LIN {X 0,Y 466.182,Z 601.705,A -85,B 0,C 180,E1 19756.767,E2 19756.767} C_VEL
LIN {X 0,Y 461.361,Z 693.458,A -85,B 0,C 180,E1 19755.037,E2 19755.037} C_VEL
LIN {X 0,Y 459.117,Z 717.943,A -85,B 0,C 180,E1 19754.37,E2 19754.37} C_VEL
LIN {X 0,Y 456.209,Z 743.457,A -85,B 0,C 180,E1 19753.448,E2 19753.448} C_VEL
LIN {X 0,Y 453.173,Z 765.825,A -85,B 0,C 180,E1 19752.424,E2 19752.424} C_VEL
LIN {X 0,Y 449.498,Z 789.387,A -85,B 0,C 180,E1 19751.096,E2 19751.096} C_VEL
LIN {X 0,Y 445.801,Z 811.052,A -85,B 0,C 180,E1 19749.642,E2 19749.642} C_VEL
LIN {X 0,Y 441.915,Z 831.707,A -85,B 0,C 180,E1 19747.983,E2 19747.983} C_VEL
LIN {X 0,Y 437.866,Z 852.231,A -85,B 0,C 180,E1 19746.062,E2 19746.062} C_VEL
LIN {X 0,Y 434.211,Z 870.106,A -85,B 0,C 180,E1 19744.106,E2 19744.106} C_VEL
LIN {X 0,Y 430.262,Z 889.208,A -85,B 0,C 180,E1 19741.682,E2 19741.682} C_VEL
LIN {X 0,Y 426.966,Z 905.358,A -85,B 0,C 180,E1 19739.304,E2 19739.304} C_VEL
LIN {X 0,Y 423.914,Z 920.881,A -85,B 0,C 180,E1 19736.625,E2 19736.625} C_VEL
LIN {X 0,Y 421.465,Z 934.402,A -85,B 0,C 180,E1 19733.934,E2 19733.934} C_VEL
LIN {X 0,Y 419.512,Z 946.432,A -85,B 0,C 180,E1 19731.094,E2 19731.094} C_VEL
LIN {X 0,Y 418.139,Z 956.77,A -85,B 0,C 180,E1 19728.256,E2 19728.256} C_VEL
LIN {X 0,Y 417.219,Z 965.635,A -85,B 0,C 180,E1 19725.285,E2 19725.285} C_VEL
LIN {X 0,Y 416.734,Z 972.905,A -85,B 0,C 180,E1 19722.33,E2 19722.33} C_VEL
LIN {X 0,Y 416.585,Z 978.694,A -85,B 0,C 180,E1 19719.254,E2 19719.254} C_VEL
LIN {X 0,Y 416.629,Z 982.359,A -85,B 0,C 180,E1 19716.615,E2 19716.615} C_VEL
LIN {X 0,Y 416.736,Z 985.143,A -85,B 0,C 180,E1 19713.577,E2 19713.577} C_VEL
LIN {X 0,Y 416.795,Z 986.147,A -85,B 0,C 180,E1 19710.687,E2 19710.687} C_VEL
LIN {X 0,Y 416.792,Z 985.858,A -85,B 0,C 180,E1 19708.075,E2 19708.075} C_VEL
LIN {X 0,Y 416.657,Z 984.108,A -85,B 0,C 180,E1 19705.044,E2 19705.044} C_VEL
LIN {X 0,Y 416.576,Z 980.619,A -85,B 0,C 180,E1 19701.997,E2 19701.997} C_VEL
LIN {X 0,Y 416.588,Z 976.376,A -85,B 0,C 180,E1 19699.35,E2 19699.35} C_VEL
LIN {X 0,Y 416.89,Z 969.637,A -85,B 0,C 180,E1 19696.122,E2 19696.122} C_VEL
LIN {X 0,Y 417.582,Z 961.789,A -85,B 0,C 180,E1 19693.158,E2 19693.158} C_VEL
LIN {X 0,Y 418.851,Z 951.921,A -85,B 0,C 180,E1 19690.039,E2 19690.039} C_VEL
LIN {X 0,Y 420.695,Z 940.588,A -85,B 0,C 180,E1 19687.059,E2 19687.059} C_VEL
LIN {X 0,Y 423.28,Z 927.489,A -85,B 0,C 180,E1 19684.086,E2 19684.086} C_VEL
LIN {X 0,Y 426.486,Z 912.889,A -85,B 0,C 180,E1 19681.264,E2 19681.264} C_VEL
LIN {X 0,Y 430.666,Z 895.41,A -85,B 0,C 180,E1 19678.351,E2 19678.351} C_VEL
LIN {X 0,Y 435.032,Z 878.269,A -85,B 0,C 180,E1 19675.888,E2 19675.888} C_VEL
LIN {X 0,Y 439.906,Z 859.257,A -85,B 0,C 180,E1 19673.539,E2 19673.539} C_VEL
LIN {X 0,Y 445.064,Z 839.529,A -85,B 0,C 180,E1 19671.428,E2 19671.428} C_VEL
LIN {X 0,Y 450.442,Z 818.443,A -85,B 0,C 180,E1 19669.512,E2 19669.512} C_VEL
LIN {X 0,Y 455.993,Z 795.957,A -85,B 0,C 180,E1 19667.772,E2 19667.772} C_VEL
LIN {X 0,Y 461.455,Z 772.834,A -85,B 0,C 180,E1 19666.273,E2 19666.273} C_VEL
LIN {X 0,Y 466.711,Z 748.74,A -85,B 0,C 180,E1 19664.991,E2 19664.991} C_VEL
LIN {X 0,Y 471.508,Z 724.263,A -85,B 0,C 180,E1 19663.949,E2 19663.949} C_VEL
LIN {X 0,Y 476.08,Z 697.875,A -85,B 0,C 180,E1 19663.088,E2 19663.088} C_VEL
LIN {X 0,Y 481.22,Z 660.217,A -85,B 0,C 180,E1 19662.172,E2 19662.172} C_VEL
LIN {X 0,Y 489.533,Z 604.335,A -85,B 0,C 180,E1 19660.843,E2 19660.843} C_VEL
LIN {X 0,Y 500.202,Z 547.443,A -85,B 0,C 180,E1 19659.451,E2 19659.451} C_VEL
LIN {X 0,Y 508.93,Z 508.11,A -85,B 0,C 180,E1 19658.468,E2 19658.468} C_VEL
LIN {X 0,Y 504.603,Z 526.167,A -85,B 0,C 180,E1 19657.559,E2 19657.559} C_VEL
LIN {X 0,Y 481.706,Z 630.182,A -85,B 0,C 180,E1 19654.492,E2 19654.492} C_VEL
LIN {X 0,Y 469.101,Z 693.847,A -85,B 0,C 180,E1 19652.444,E2 19652.444} C_VEL
LIN {X 0,Y 463.766,Z 717.456,A -85,B 0,C 180,E1 19651.45,E2 19651.45} C_VEL
LIN {X 0,Y 458.09,Z 740.922,A -85,B 0,C 180,E1 19650.185,E2 19650.185} C_VEL
LIN {X 0,Y 452.388,Z 763.754,A -85,B 0,C 180,E1 19648.661,E2 19648.661} C_VEL
LIN {X 0,Y 447.011,Z 785.108,A -85,B 0,C 180,E1 19646.934,E2 19646.934} C_VEL
LIN {X 0,Y 442.238,Z 804.171,A -85,B 0,C 180,E1 19645.083,E2 19645.083} C_VEL
LIN {X 0,Y 437.83,Z 821.686,A -85,B 0,C 180,E1 19643.058,E2 19643.058} C_VEL
LIN {X 0,Y 433.913,Z 837.047,A -85,B 0,C 180,E1 19640.927,E2 19640.927} C_VEL
LIN {X 0,Y 430.445,Z 850.31,A -85,B 0,C 180,E1 19638.697,E2 19638.697} C_VEL
LIN {X 0,Y 427.606,Z 860.933,A -85,B 0,C 180,E1 19636.519,E2 19636.519} C_VEL
LIN {X 0,Y 425.193,Z 869.743,A -85,B 0,C 180,E1 19634.295,E2 19634.295} C_VEL
LIN {X 0,Y 423.039,Z 877.204,A -85,B 0,C 180,E1 19631.867,E2 19631.867} C_VEL
LIN {X 0,Y 421.42,Z 882.367,A -85,B 0,C 180,E1 19629.56,E2 19629.56} C_VEL
LIN {X 0,Y 420.191,Z 885.911,A -85,B 0,C 180,E1 19627.245,E2 19627.245} C_VEL
LIN {X 0,Y 419.213,Z 887.887,A -85,B 0,C 180,E1 19624.789,E2 19624.789} C_VEL
LIN {X 0,Y 418.581,Z 888.17,A -85,B 0,C 180,E1 19622.464,E2 19622.464} C_VEL
LIN {X 0,Y 418.161,Z 886.727,A -85,B 0,C 180,E1 19620,E2 19620} C_VEL
LIN {X 0,Y 417.948,Z 883.54,A -85,B 0,C 180,E1 19617.532,E2 19617.532} C_VEL
LIN {X 0,Y 417.955,Z 878.555,A -85,B 0,C 180,E1 19615.059,E2 19615.059} C_VEL
LIN {X 0,Y 418.197,Z 871.701,A -85,B 0,C 180,E1 19612.582,E2 19612.582} C_VEL
LIN {X 0,Y 418.711,Z 862.825,A -85,B 0,C 180,E1 19610.099,E2 19610.099} C_VEL
LIN {X 0,Y 419.516,Z 852.331,A -85,B 0,C 180,E1 19607.745,E2 19607.745} C_VEL
LIN {X 0,Y 420.579,Z 840.438,A -85,B 0,C 180,E1 19605.544,E2 19605.544} C_VEL
LIN {X 0,Y 421.988,Z 826.127,A -85,B 0,C 180,E1 19603.339,E2 19603.339} C_VEL
LIN {X 0,Y 423.658,Z 810.108,A -85,B 0,C 180,E1 19601.278,E2 19601.278} C_VEL
LIN {X 0,Y 425.556,Z 792.28,A -85,B 0,C 180,E1 19599.363,E2 19599.363} C_VEL
LIN {X 0,Y 427.535,Z 773.248,A -85,B 0,C 180,E1 19597.663,E2 19597.663} C_VEL
LIN {X 0,Y 429.463,Z 754.068,A -85,B 0,C 180,E1 19596.247,E2 19596.247} C_VEL
LIN {X 0,Y 431.425,Z 733.007,A -85,B 0,C 180,E1 19594.986,E2 19594.986} C_VEL
LIN {X 0,Y 433.222,Z 711.178,A -85,B 0,C 180,E1 19593.953,E2 19593.953} C_VEL
LIN {X 0,Y 434.895,Z 687.679,A -85,B 0,C 180,E1 19593.121,E2 19593.121} C_VEL
LIN {X 0,Y 437.042,Z 646.566,A -85,B 0,C 180,E1 19592.122,E2 19592.122} C_VEL
LIN {X 0,Y 444.712,Z 506.021,A -85,B 0,C 180,E1 19588.907,E2 19588.907} C_VEL
LIN {X 0,Y 439.779,Z 438.733,A -85,B 0,C 180,E1 19586.694,E2 19586.694} C_VEL
LIN {X 0,Y 445.969,Z 387.644,A -85,B 0,C 180,E1 19582.511,E2 19582.511} C_VEL
LIN {X 0,Y 451.691,Z 344.172,A -85,B 0,C 180,E1 19578.936,E2 19578.936} C_VEL
LIN {X 0,Y 453.675,Z 344.144,A -85,B 0,C 180,E1 19578.609,E2 19578.609} C_VEL
LIN {X 0,Y 456.593,Z 342.501,A -85,B 0,C 180,E1 19578.262,E2 19578.262} C_VEL
LIN {X 0,Y 459.898,Z 339.563,A -85,B 0,C 180,E1 19577.96,E2 19577.96} C_VEL
LIN {X 0,Y 463.43,Z 338.215,A -85,B 0,C 180,E1 19577.52,E2 19577.52} C_VEL
LIN {X 0,Y 468.257,Z 334.771,A -85,B 0,C 180,E1 19577.064,E2 19577.064} C_VEL
LIN {X 0,Y 472.208,Z 333.263,A -85,B 0,C 180,E1 19576.6,E2 19576.6} C_VEL
LIN {X 0,Y 476.586,Z 346.018,A -85,B 0,C 180,E1 19574.994,E2 19574.994} C_VEL
LIN {X 0,Y 476.081,Z 370.363,A -85,B 0,C 180,E1 19573.293,E2 19573.293} C_VEL
LIN {X 0,Y 470.702,Z 395.368,A -85,B 0,C 180,E1 19572.381,E2 19572.381} C_VEL
LIN {X 0,Y 466.885,Z 477.849,A -85,B 0,C 180,E1 19571.021,E2 19571.021} C_VEL
LIN {X 0,Y 462.789,Z 540.682,A -85,B 0,C 180,E1 19569.779,E2 19569.779} C_VEL
LIN {X 0,Y 457.359,Z 607.896,A -85,B 0,C 180,E1 19568.227,E2 19568.227} C_VEL
LIN {X 0,Y 453.808,Z 652.838,A -85,B 0,C 180,E1 19567.008,E2 19567.008} C_VEL
LIN {X 0,Y 452.145,Z 676.013,A -85,B 0,C 180,E1 19566.219,E2 19566.219} C_VEL
LIN {X 0,Y 450.073,Z 696.948,A -85,B 0,C 180,E1 19565.284,E2 19565.284} C_VEL
LIN {X 0,Y 447.372,Z 718.396,A -85,B 0,C 180,E1 19564.073,E2 19564.073} C_VEL
LIN {X 0,Y 444.251,Z 739.171,A -85,B 0,C 180,E1 19562.619,E2 19562.619} C_VEL
LIN {X 0,Y 440.936,Z 758.361,A -85,B 0,C 180,E1 19560.992,E2 19560.992} C_VEL
LIN {X 0,Y 438.931,Z 764.725,A -85,B 0,C 180,E1 19560.467,E2 19560.467} C_VEL
LIN {X 0,Y 430.735,Z 780.584,A -85,B 0,C 180,E1 19559.246,E2 19559.246} C_VEL
LIN {X 0,Y 428.649,Z 786.403,A -85,B 0,C 180,E1 19558.626,E2 19558.626} C_VEL
LIN {X 0,Y 425.203,Z 802.108,A -85,B 0,C 180,E1 19556.538,E2 19556.538} C_VEL
LIN {X 0,Y 421.843,Z 816.908,A -85,B 0,C 180,E1 19554.209,E2 19554.209} C_VEL
LIN {X 0,Y 418.786,Z 830.224,A -85,B 0,C 180,E1 19551.72,E2 19551.72} C_VEL
LIN {X 0,Y 415.99,Z 842.599,A -85,B 0,C 180,E1 19548.935,E2 19548.935} C_VEL
LIN {X 0,Y 413.787,Z 852.799,A -85,B 0,C 180,E1 19546.134,E2 19546.134} C_VEL
LIN {X 0,Y 412.078,Z 861.435,A -85,B 0,C 180,E1 19543.185,E2 19543.185} C_VEL
LIN {X 0,Y 410.917,Z 867.862,A -85,B 0,C 180,E1 19540.374,E2 19540.374} C_VEL
LIN {X 0,Y 410.156,Z 872.891,A -85,B 0,C 180,E1 19537.424,E2 19537.424} C_VEL
LIN {X 0,Y 409.729,Z 876.243,A -85,B 0,C 180,E1 19534.479,E2 19534.479} C_VEL
LIN {X 0,Y 409.54,Z 877.981,A -85,B 0,C 180,E1 19531.539,E2 19531.539} C_VEL
LIN {X 0,Y 409.523,Z 878.039,A -85,B 0,C 180,E1 19528.741,E2 19528.741} C_VEL
LIN {X 0,Y 409.692,Z 876.537,A -85,B 0,C 180,E1 19525.801,E2 19525.801} C_VEL
LIN {X 0,Y 410.094,Z 873.424,A -85,B 0,C 180,E1 19522.857,E2 19522.857} C_VEL
LIN {X 0,Y 410.768,Z 868.937,A -85,B 0,C 180,E1 19520.048,E2 19520.048} C_VEL
LIN {X 0,Y 411.91,Z 862.424,A -85,B 0,C 180,E1 19517.096,E2 19517.096} C_VEL
LIN {X 0,Y 413.462,Z 854.365,A -85,B 0,C 180,E1 19514.26,E2 19514.26} C_VEL
LIN {X 0,Y 415.547,Z 844.595,A -85,B 0,C 180,E1 19511.481,E2 19511.481} C_VEL
LIN {X 0,Y 418.086,Z 833.296,A -85,B 0,C 180,E1 19508.83,E2 19508.83} C_VEL
LIN {X 0,Y 421.02,Z 820.573,A -85,B 0,C 180,E1 19506.337,E2 19506.337} C_VEL
LIN {X 0,Y 424.266,Z 806.441,A -85,B 0,C 180,E1 19504.001,E2 19504.001} C_VEL
LIN {X 0,Y 427.748,Z 790.854,A -85,B 0,C 180,E1 19501.824,E2 19501.824} C_VEL
LIN {X 0,Y 431.38,Z 773.694,A -85,B 0,C 180,E1 19499.803,E2 19499.803} C_VEL
LIN {X 0,Y 434.929,Z 755.568,A -85,B 0,C 180,E1 19498.008,E2 19498.008} C_VEL
LIN {X 0,Y 438.301,Z 736.243,A -85,B 0,C 180,E1 19496.412,E2 19496.412} C_VEL
LIN {X 0,Y 441.375,Z 715.92,A -85,B 0,C 180,E1 19495.03,E2 19495.03} C_VEL
LIN {X 0,Y 443.968,Z 695.234,A -85,B 0,C 180,E1 19493.891,E2 19493.891} C_VEL
LIN {X 0,Y 446.008,Z 674.403,A -85,B 0,C 180,E1 19492.983,E2 19492.983} C_VEL
LIN {X 0,Y 447.966,Z 647.329,A -85,B 0,C 180,E1 19492.093,E2 19492.093} C_VEL
LIN {X 0,Y 452.25,Z 596.981,A -85,B 0,C 180,E1 19490.753,E2 19490.753} C_VEL
LIN {X 0,Y 457.54,Z 531.945,A -85,B 0,C 180,E1 19489.27,E2 19489.27} C_VEL
LIN {X 0,Y 461.65,Z 467.541,A -85,B 0,C 180,E1 19488.024,E2 19488.024} C_VEL
LIN {X 0,Y 465.122,Z 396.05,A -85,B 0,C 180,E1 19486.831,E2 19486.831} C_VEL
LIN {X 0,Y 470.511,Z 371.711,A -85,B 0,C 180,E1 19485.914,E2 19485.914} C_VEL
LIN {X 0,Y 470.855,Z 349.322,A -85,B 0,C 180,E1 19484.319,E2 19484.319} C_VEL
LIN {X 0,Y 463.855,Z 330.038,A -85,B 0,C 180,E1 19481.766,E2 19481.766} C_VEL
LIN {X 0,Y 456.491,Z 312.145,A -85,B 0,C 180,E1 19479.112,E2 19479.112} C_VEL
LIN {X 0,Y 448.714,Z 295.881,A -85,B 0,C 180,E1 19476.445,E2 19476.445} C_VEL
LIN {X 0,Y 441.192,Z 281.498,A -85,B 0,C 180,E1 19473.806,E2 19473.806} C_VEL
LIN {X 0,Y 434.542,Z 270.327,A -85,B 0,C 180,E1 19471.489,E2 19471.489} C_VEL
LIN {X 0,Y 429.661,Z 262.251,A -85,B 0,C 180,E1 19469.715,E2 19469.715} C_VEL
LIN {X 0,Y 426.904,Z 258.059,A -85,B 0,C 180,E1 19468.695,E2 19468.695} C_VEL
LIN {X 0,Y 423.194,Z 252.399,A -85,B 0,C 180,E1 19467.282,E2 19467.282} C_VEL
LIN {X 0,Y 419.793,Z 247.902,A -85,B 0,C 180,E1 19465.993,E2 19465.993} C_VEL
LIN {X 0,Y 418.942,Z 246.069,A -85,B 0,C 180,E1 19465.594,E2 19465.594} C_VEL
LIN {X 0,Y 416.059,Z 242.908,A -85,B 0,C 180,E1 19464.492,E2 19464.492} C_VEL
LIN {X 0,Y 414.671,Z 240.056,A -85,B 0,C 180,E1 19463.822,E2 19463.822} C_VEL
LIN {X 0,Y 411.827,Z 237.422,A -85,B 0,C 180,E1 19462.709,E2 19462.709} C_VEL
LIN {X 0,Y 410.633,Z 234.295,A -85,B 0,C 180,E1 19462.024,E2 19462.024} C_VEL
LIN {X 0,Y 410.594,Z 234.03,A -85,B 0,C 180,E1 19458.162,E2 19458.162} C_VEL
LIN {X 0,Y 410.604,Z 234.058,A -85,B 0,C 180,E1 19454.238,E2 19454.238} C_VEL
LIN {X 0,Y 410.596,Z 234.057,A -85,B 0,C 180,E1 19450.24,E2 19450.24} C_VEL
LIN {X 0,Y 410.596,Z 234.027,A -85,B 0,C 180,E1 19446.291,E2 19446.291} C_VEL
LIN {X 0,Y 410.601,Z 234.083,A -85,B 0,C 180,E1 19442.373,E2 19442.373} C_VEL
LIN {X 0,Y 410.597,Z 234.031,A -85,B 0,C 180,E1 19438.465,E2 19438.465} C_VEL
LIN {X 0,Y 410.599,Z 234.046,A -85,B 0,C 180,E1 19434.55,E2 19434.55} C_VEL
LIN {X 0,Y 410.602,Z 234.061,A -85,B 0,C 180,E1 19430.61,E2 19430.61} C_VEL
LIN {X 0,Y 410.605,Z 234.083,A -85,B 0,C 180,E1 19426.624,E2 19426.624} C_VEL
LIN {X 0,Y 410.601,Z 234.084,A -85,B 0,C 180,E1 19422.717,E2 19422.717} C_VEL
LIN {X 0,Y 410.633,Z 234.282,A -85,B 0,C 180,E1 19422.462,E2 19422.462} C_VEL
LIN {X 0,Y 411.874,Z 237.541,A -85,B 0,C 180,E1 19421.75,E2 19421.75} C_VEL
LIN {X 0,Y 413.191,Z 239.4,A -85,B 0,C 180,E1 19421.225,E2 19421.225} C_VEL
LIN {X 0,Y 415.204,Z 243.299,A -85,B 0,C 180,E1 19420.297,E2 19420.297} C_VEL
LIN {X 0,Y 420.886,Z 254.249,A -85,B 0,C 180,E1 19417.807,E2 19417.807} C_VEL
LIN {X 0,Y 427.8,Z 267.468,A -85,B 0,C 180,E1 19414.973,E2 19414.973} C_VEL
LIN {X 0,Y 436.306,Z 284.141,A -85,B 0,C 180,E1 19411.68,E2 19411.68} C_VEL
LIN {X 0,Y 446.297,Z 304.362,A -85,B 0,C 180,E1 19408.08,E2 19408.08} C_VEL
LIN {X 0,Y 456.718,Z 326.072,A -85,B 0,C 180,E1 19404.634,E2 19404.634} C_VEL
LIN {X 0,Y 474.355,Z 353.885,A -85,B 0,C 180,E1 19402.032,E2 19402.032} C_VEL
LIN {X 0,Y 474.205,Z 360.312,A -85,B 0,C 180,E1 19401.883,E2 19401.883} C_VEL
LIN {X 0,Y 459.21,Z 606.522,A -85,B 0,C 180,E1 19397.216,E2 19397.216} C_VEL
LIN {X 0,Y 454.457,Z 693.43,A -85,B 0,C 180,E1 19395.543,E2 19395.543} C_VEL
LIN {X 0,Y 452.163,Z 717.773,A -85,B 0,C 180,E1 19394.869,E2 19394.869} C_VEL
LIN {X 0,Y 449.295,Z 742.351,A -85,B 0,C 180,E1 19393.975,E2 19393.975} C_VEL
LIN {X 0,Y 446.278,Z 764.081,A -85,B 0,C 180,E1 19392.975,E2 19392.975} C_VEL
LIN {X 0,Y 442.507,Z 787.894,A -85,B 0,C 180,E1 19391.63,E2 19391.63} C_VEL
LIN {X 0,Y 438.714,Z 809.559,A -85,B 0,C 180,E1 19390.165,E2 19390.165} C_VEL
LIN {X 0,Y 434.774,Z 830.163,A -85,B 0,C 180,E1 19388.501,E2 19388.501} C_VEL
LIN {X 0,Y 430.744,Z 850.203,A -85,B 0,C 180,E1 19386.625,E2 19386.625} C_VEL
LIN {X 0,Y 426.766,Z 869.103,A -85,B 0,C 180,E1 19384.541,E2 19384.541} C_VEL
LIN {X 0,Y 422.811,Z 887.794,A -85,B 0,C 180,E1 19382.147,E2 19382.147} C_VEL
LIN {X 0,Y 419.509,Z 903.423,A -85,B 0,C 180,E1 19379.82,E2 19379.82} C_VEL
LIN {X 0,Y 416.377,Z 918.925,A -85,B 0,C 180,E1 19377.146,E2 19377.146} C_VEL
LIN {X 0,Y 413.922,Z 931.913,A -85,B 0,C 180,E1 19374.55,E2 19374.55} C_VEL
LIN {X 0,Y 411.744,Z 944.833,A -85,B 0,C 180,E1 19371.512,E2 19371.512} C_VEL
LIN {X 0,Y 410.284,Z 955.269,A -85,B 0,C 180,E1 19368.618,E2 19368.618} C_VEL
LIN {X 0,Y 409.272,Z 964.688,A -85,B 0,C 180,E1 19365.444,E2 19365.444} C_VEL
LIN {X 0,Y 408.776,Z 971.983,A -85,B 0,C 180,E1 19362.43,E2 19362.43} C_VEL
LIN {X 0,Y 408.629,Z 977.786,A -85,B 0,C 180,E1 19359.294,E2 19359.294} C_VEL
LIN {X 0,Y 408.681,Z 981.444,A -85,B 0,C 180,E1 19356.603,E2 19356.603} C_VEL
LIN {X 0,Y 408.797,Z 984.212,A -85,B 0,C 180,E1 19353.506,E2 19353.506} C_VEL
LIN {X 0,Y 408.855,Z 985.183,A -85,B 0,C 180,E1 19350.56,E2 19350.56} C_VEL
LIN {X 0,Y 408.837,Z 984.862,A -85,B 0,C 180,E1 19347.898,E2 19347.898} C_VEL
LIN {X 0,Y 408.69,Z 983.057,A -85,B 0,C 180,E1 19344.806,E2 19344.806} C_VEL
LIN {X 0,Y 408.594,Z 979.51,A -85,B 0,C 180,E1 19341.698,E2 19341.698} C_VEL
LIN {X 0,Y 408.613,Z 975.041,A -85,B 0,C 180,E1 19338.892,E2 19338.892} C_VEL
LIN {X 0,Y 408.992,Z 968.066,A -85,B 0,C 180,E1 19335.56,E2 19335.56} C_VEL
LIN {X 0,Y 409.782,Z 960.115,A -85,B 0,C 180,E1 19332.535,E2 19332.535} C_VEL
LIN {X 0,Y 411.287,Z 949.569,A -85,B 0,C 180,E1 19329.21,E2 19329.21} C_VEL
LIN {X 0,Y 413.253,Z 938.67,A -85,B 0,C 180,E1 19326.319,E2 19326.319} C_VEL
LIN {X 0,Y 416.402,Z 923.909,A -85,B 0,C 180,E1 19322.983,E2 19322.983} C_VEL
LIN {X 0,Y 419.914,Z 909.28,A -85,B 0,C 180,E1 19320.154,E2 19320.154} C_VEL
LIN {X 0,Y 424.304,Z 892.298,A -85,B 0,C 180,E1 19317.34,E2 19317.34} C_VEL
LIN {X 0,Y 429.296,Z 873.956,A -85,B 0,C 180,E1 19314.716,E2 19314.716} C_VEL
LIN {X 0,Y 434.639,Z 854.657,A -85,B 0,C 180,E1 19312.354,E2 19312.354} C_VEL
LIN {X 0,Y 440.371,Z 833.928,A -85,B 0,C 180,E1 19310.186,E2 19310.186} C_VEL
LIN {X 0,Y 445.99,Z 813.441,A -85,B 0,C 180,E1 19308.337,E2 19308.337} C_VEL
LIN {X 0,Y 451.965,Z 790.62,A -85,B 0,C 180,E1 19306.613,E2 19306.613} C_VEL
LIN {X 0,Y 457.815,Z 767.151,A -85,B 0,C 180,E1 19305.134,E2 19305.134} C_VEL
LIN {X 0,Y 463.428,Z 743.115,A -85,B 0,C 180,E1 19303.893,E2 19303.893} C_VEL
LIN {X 0,Y 468.675,Z 718.317,A -85,B 0,C 180,E1 19302.875,E2 19302.875} C_VEL
LIN {X 0,Y 473.177,Z 693.617,A -85,B 0,C 180,E1 19302.1,E2 19302.1} C_VEL
LIN {X 0,Y 485.132,Z 617.626,A -85,B 0,C 180,E1 19300.249,E2 19300.249} C_VEL
LIN {X 0,Y 496.148,Z 562.189,A -85,B 0,C 180,E1 19298.884,E2 19298.884} C_VEL
LIN {X 0,Y 502.171,Z 535.812,A -85,B 0,C 180,E1 19298.223,E2 19298.223} C_VEL
LIN {X 0,Y 478.06,Z 639.781,A -85,B 0,C 180,E1 19295.149,E2 19295.149} C_VEL
LIN {X 0,Y 466.558,Z 693.913,A -85,B 0,C 180,E1 19293.393,E2 19293.393} C_VEL
LIN {X 0,Y 460.795,Z 717.287,A -85,B 0,C 180,E1 19292.41,E2 19292.41} C_VEL
LIN {X 0,Y 454.74,Z 739.998,A -85,B 0,C 180,E1 19291.186,E2 19291.186} C_VEL
LIN {X 0,Y 448.459,Z 762.678,A -85,B 0,C 180,E1 19289.668,E2 19289.668} C_VEL
LIN {X 0,Y 442.189,Z 785.109,A -85,B 0,C 180,E1 19287.836,E2 19287.836} C_VEL
LIN {X 0,Y 436.82,Z 804.476,A -85,B 0,C 180,E1 19285.926,E2 19285.926} C_VEL
LIN {X 0,Y 432.024,Z 821.806,A -85,B 0,C 180,E1 19283.893,E2 19283.893} C_VEL
LIN {X 0,Y 427.866,Z 836.688,A -85,B 0,C 180,E1 19281.813,E2 19281.813} C_VEL
LIN {X 0,Y 424.085,Z 850.143,A -85,B 0,C 180,E1 19279.561,E2 19279.561} C_VEL
LIN {X 0,Y 420.685,Z 861.897,A -85,B 0,C 180,E1 19277.141,E2 19277.141} C_VEL
LIN {X 0,Y 417.846,Z 871.334,A -85,B 0,C 180,E1 19274.694,E2 19274.694} C_VEL
LIN {X 0,Y 415.638,Z 878.281,A -85,B 0,C 180,E1 19272.363,E2 19272.363} C_VEL
LIN {X 0,Y 413.877,Z 883.502,A -85,B 0,C 180,E1 19270.017,E2 19270.017} C_VEL
LIN {X 0,Y 412.447,Z 887.202,A -85,B 0,C 180,E1 19267.522,E2 19267.522} C_VEL
LIN {X 0,Y 411.394,Z 889.136,A -85,B 0,C 180,E1 19265.02,E2 19265.02} C_VEL
LIN {X 0,Y 410.666,Z 889.291,A -85,B 0,C 180,E1 19262.512,E2 19262.512} C_VEL
LIN {X 0,Y 410.24,Z 887.847,A -85,B 0,C 180,E1 19260.14,E2 19260.14} C_VEL
LIN {X 0,Y 410.002,Z 884.604,A -85,B 0,C 180,E1 19257.624,E2 19257.624} C_VEL
LIN {X 0,Y 409.997,Z 879.569,A -85,B 0,C 180,E1 19255.103,E2 19255.103} C_VEL
LIN {X 0,Y 410.237,Z 872.646,A -85,B 0,C 180,E1 19252.578,E2 19252.578} C_VEL
LIN {X 0,Y 410.759,Z 863.693,A -85,B 0,C 180,E1 19250.047,E2 19250.047} C_VEL
LIN {X 0,Y 411.582,Z 853.184,A -85,B 0,C 180,E1 19247.656,E2 19247.656} C_VEL
LIN {X 0,Y 412.682,Z 841.23,A -85,B 0,C 180,E1 19245.405,E2 19245.405} C_VEL
LIN {X 0,Y 414.082,Z 827.361,A -85,B 0,C 180,E1 19243.228,E2 19243.228} C_VEL
LIN {X 0,Y 415.785,Z 811.363,A -85,B 0,C 180,E1 19241.128,E2 19241.128} C_VEL
LIN {X 0,Y 417.725,Z 793.581,A -85,B 0,C 180,E1 19239.178,E2 19239.178} C_VEL
LIN {X 0,Y 419.747,Z 774.635,A -85,B 0,C 180,E1 19237.448,E2 19237.448} C_VEL
LIN {X 0,Y 421.818,Z 754.622,A -85,B 0,C 180,E1 19235.939,E2 19235.939} C_VEL
LIN {X 0,Y 423.846,Z 733.462,A -85,B 0,C 180,E1 19234.648,E2 19234.648} C_VEL
LIN {X 0,Y 425.613,Z 712.677,A -85,B 0,C 180,E1 19233.639,E2 19233.639} C_VEL
LIN {X 0,Y 427.276,Z 690.14,A -85,B 0,C 180,E1 19232.808,E2 19232.808} C_VEL
LIN {X 0,Y 429.095,Z 657.974,A -85,B 0,C 180,E1 19231.976,E2 19231.976} C_VEL
LIN {X 0,Y 437.616,Z 506.725,A -85,B 0,C 180,E1 19228.426,E2 19228.426} C_VEL
LIN {X 0,Y 432.779,Z 437.458,A -85,B 0,C 180,E1 19226.085,E2 19226.085} C_VEL
LIN {X 0,Y 439.247,Z 386.125,A -85,B 0,C 180,E1 19221.827,E2 19221.827} C_VEL
LIN {X 0,Y 443.283,Z 356.55,A -85,B 0,C 180,E1 19219.359,E2 19219.359} C_VEL
LIN {X 0,Y 445.261,Z 356.47,A -85,B 0,C 180,E1 19219.025,E2 19219.025} C_VEL
LIN {X 0,Y 448.955,Z 354.156,A -85,B 0,C 180,E1 19218.588,E2 19218.588} C_VEL
LIN {X 0,Y 451.823,Z 351.613,A -85,B 0,C 180,E1 19218.317,E2 19218.317} C_VEL
LIN {X 0,Y 455.703,Z 349.897,A -85,B 0,C 180,E1 19217.823,E2 19217.823} C_VEL
LIN {X 0,Y 460.446,Z 346.36,A -85,B 0,C 180,E1 19217.349,E2 19217.349} C_VEL
LIN {X 0,Y 465.632,Z 343.618,A -85,B 0,C 180,E1 19216.763,E2 19216.763} C_VEL
LIN {X 0,Y 468.15,Z 341.884,A -85,B 0,C 180,E1 19216.527,E2 19216.527} C_VEL
LIN {X 0,Y 470.899,Z 349.839,A -85,B 0,C 180,E1 19215.516,E2 19215.516} C_VEL
LIN {X 0,Y 470.365,Z 372.226,A -85,B 0,C 180,E1 19213.953,E2 19213.953} C_VEL
LIN {X 0,Y 464.775,Z 398.05,A -85,B 0,C 180,E1 19213.014,E2 19213.014} C_VEL
LIN {X 0,Y 460.852,Z 480.196,A -85,B 0,C 180,E1 19211.649,E2 19211.649} C_VEL
LIN {X 0,Y 456.69,Z 542.095,A -85,B 0,C 180,E1 19210.412,E2 19210.412} C_VEL
LIN {X 0,Y 451.226,Z 607.78,A -85,B 0,C 180,E1 19208.878,E2 19208.878} C_VEL
LIN {X 0,Y 447.491,Z 653.023,A -85,B 0,C 180,E1 19207.635,E2 19207.635} C_VEL
LIN {X 0,Y 445.668,Z 677.543,A -85,B 0,C 180,E1 19206.792,E2 19206.792} C_VEL
LIN {X 0,Y 443.448,Z 699.052,A -85,B 0,C 180,E1 19205.812,E2 19205.812} C_VEL
LIN {X 0,Y 440.746,Z 719.67,A -85,B 0,C 180,E1 19204.628,E2 19204.628} C_VEL
LIN {X 0,Y 437.713,Z 739.284,A -85,B 0,C 180,E1 19203.247,E2 19203.247} C_VEL
LIN {X 0,Y 434.389,Z 758.036,A -85,B 0,C 180,E1 19201.656,E2 19201.656} C_VEL
LIN {X 0,Y 430.869,Z 775.879,A -85,B 0,C 180,E1 19199.853,E2 19199.853} C_VEL
LIN {X 0,Y 428.649,Z 786.403,A -85,B 0,C 180,E1 19198.626,E2 19198.626} C_VEL
LIN {X 0,Y 426.569,Z 792.199,A -85,B 0,C 180,E1 19197.982,E2 19197.982} C_VEL
LIN {X 0,Y 418.163,Z 806.503,A -85,B 0,C 180,E1 19196.446,E2 19196.446} C_VEL
LIN {X 0,Y 416.054,Z 811.677,A -85,B 0,C 180,E1 19195.707,E2 19195.707} C_VEL
LIN {X 0,Y 412.727,Z 825.579,A -85,B 0,C 180,E1 19193.259,E2 19193.259} C_VEL
LIN {X 0,Y 409.828,Z 837.724,A -85,B 0,C 180,E1 19190.718,E2 19190.718} C_VEL
LIN {X 0,Y 407.198,Z 848.973,A -85,B 0,C 180,E1 19187.875,E2 19187.875} C_VEL
LIN {X 0,Y 405.09,Z 858.595,A -85,B 0,C 180,E1 19184.875,E2 19184.875} C_VEL
LIN {X 0,Y 403.628,Z 865.866,A -85,B 0,C 180,E1 19182.011,E2 19182.011} C_VEL
LIN {X 0,Y 402.636,Z 871.479,A -85,B 0,C 180,E1 19179.145,E2 19179.145} C_VEL
LIN {X 0,Y 402.009,Z 875.701,A -85,B 0,C 180,E1 19176.14,E2 19176.14} C_VEL
LIN {X 0,Y 401.697,Z 878.215,A -85,B 0,C 180,E1 19173.282,E2 19173.282} C_VEL
LIN {X 0,Y 401.58,Z 879.177,A -85,B 0,C 180,E1 19170.285,E2 19170.285} C_VEL
LIN {X 0,Y 401.639,Z 878.588,A -85,B 0,C 180,E1 19167.432,E2 19167.432} C_VEL
LIN {X 0,Y 401.919,Z 876.416,A -85,B 0,C 180,E1 19164.432,E2 19164.432} C_VEL
LIN {X 0,Y 402.47,Z 872.618,A -85,B 0,C 180,E1 19161.427,E2 19161.427} C_VEL
LIN {X 0,Y 403.427,Z 867.074,A -85,B 0,C 180,E1 19158.419,E2 19158.419} C_VEL
LIN {X 0,Y 404.801,Z 859.988,A -85,B 0,C 180,E1 19155.53,E2 19155.53} C_VEL
LIN {X 0,Y 406.685,Z 851.263,A -85,B 0,C 180,E1 19152.693,E2 19152.693} C_VEL
LIN {X 0,Y 409.166,Z 840.507,A -85,B 0,C 180,E1 19149.845,E2 19149.845} C_VEL
LIN {X 0,Y 412.106,Z 828.21,A -85,B 0,C 180,E1 19147.157,E2 19147.157} C_VEL
LIN {X 0,Y 415.446,Z 814.375,A -85,B 0,C 180,E1 19144.633,E2 19144.633} C_VEL
LIN {X 0,Y 418.979,Z 799.456,A -85,B 0,C 180,E1 19142.343,E2 19142.343} C_VEL
LIN {X 0,Y 422.616,Z 783.429,A -85,B 0,C 180,E1 19140.263,E2 19140.263} C_VEL
LIN {X 0,Y 426.273,Z 766.208,A -85,B 0,C 180,E1 19138.373,E2 19138.373} C_VEL
LIN {X 0,Y 429.954,Z 747.171,A -85,B 0,C 180,E1 19136.625,E2 19136.625} C_VEL
LIN {X 0,Y 433.345,Z 727.035,A -85,B 0,C 180,E1 19135.094,E2 19135.094} C_VEL
LIN {X 0,Y 436.271,Z 706.649,A -85,B 0,C 180,E1 19133.831,E2 19133.831} C_VEL
LIN {X 0,Y 438.733,Z 685.135,A -85,B 0,C 180,E1 19132.765,E2 19132.765} C_VEL
LIN {X 0,Y 440.593,Z 663.377,A -85,B 0,C 180,E1 19131.94,E2 19131.94} C_VEL
LIN {X 0,Y 444.033,Z 620.387,A -85,B 0,C 180,E1 19130.681,E2 19130.681} C_VEL
LIN {X 0,Y 449.713,Z 556.319,A -85,B 0,C 180,E1 19129.119,E2 19129.119} C_VEL
LIN {X 0,Y 454.399,Z 491.907,A -85,B 0,C 180,E1 19127.781,E2 19127.781} C_VEL
LIN {X 0,Y 457.906,Z 425.096,A -85,B 0,C 180,E1 19126.629,E2 19126.629} C_VEL
LIN {X 0,Y 459.25,Z 398.805,A -85,B 0,C 180,E1 19126.183,E2 19126.183} C_VEL
LIN {X 0,Y 464.899,Z 373.15,A -85,B 0,C 180,E1 19125.215,E2 19125.215} C_VEL
LIN {X 0,Y 465.39,Z 353.946,A -85,B 0,C 180,E1 19123.86,E2 19123.86} C_VEL
LIN {X 0,Y 458.648,Z 335.098,A -85,B 0,C 180,E1 19121.343,E2 19121.343} C_VEL
LIN {X 0,Y 451.385,Z 317.254,A -85,B 0,C 180,E1 19118.659,E2 19118.659} C_VEL
LIN {X 0,Y 443.902,Z 301.367,A -85,B 0,C 180,E1 19116.009,E2 19116.009} C_VEL
LIN {X 0,Y 436.447,Z 287.134,A -85,B 0,C 180,E1 19113.356,E2 19113.356} C_VEL
LIN {X 0,Y 430.532,Z 276.878,A -85,B 0,C 180,E1 19111.192,E2 19111.192} C_VEL
LIN {X 0,Y 425.367,Z 268.39,A -85,B 0,C 180,E1 19109.271,E2 19109.271} C_VEL
LIN {X 0,Y 422.017,Z 263.167,A -85,B 0,C 180,E1 19107.978,E2 19107.978} C_VEL
LIN {X 0,Y 418.72,Z 258.143,A -85,B 0,C 180,E1 19106.676,E2 19106.676} C_VEL
LIN {X 0,Y 416.109,Z 254.486,A -85,B 0,C 180,E1 19105.629,E2 19105.629} C_VEL
LIN {X 0,Y 415.045,Z 252.734,A -85,B 0,C 180,E1 19105.164,E2 19105.164} C_VEL
LIN {X 0,Y 412.308,Z 249.235,A -85,B 0,C 180,E1 19104.043,E2 19104.043} C_VEL
LIN {X 0,Y 411.215,Z 247.12,A -85,B 0,C 180,E1 19103.502,E2 19103.502} C_VEL
LIN {X 0,Y 408.325,Z 244.044,A -85,B 0,C 180,E1 19102.306,E2 19102.306} C_VEL
LIN {X 0,Y 407.098,Z 241.256,A -85,B 0,C 180,E1 19101.618,E2 19101.618} C_VEL
LIN {X 0,Y 404.13,Z 238.776,A -85,B 0,C 180,E1 19100.342,E2 19100.342} C_VEL
LIN {X 0,Y 402.797,Z 235.839,A -85,B 0,C 180,E1 19099.542,E2 19099.542} C_VEL
LIN {X 0,Y 402.657,Z 235.03,A -85,B 0,C 180,E1 19099.33,E2 19099.33} C_VEL
LIN {X 0,Y 402.661,Z 235.068,A -85,B 0,C 180,E1 19095.409,E2 19095.409} C_VEL
LIN {X 0,Y 402.647,Z 235.02,A -85,B 0,C 180,E1 19091.459,E2 19091.459} C_VEL
LIN {X 0,Y 402.645,Z 235.035,A -85,B 0,C 180,E1 19087.563,E2 19087.563} C_VEL
LIN {X 0,Y 402.646,Z 235.058,A -85,B 0,C 180,E1 19083.559,E2 19083.559} C_VEL
LIN {X 0,Y 402.64,Z 235.014,A -85,B 0,C 180,E1 19079.573,E2 19079.573} C_VEL
LIN {X 0,Y 402.644,Z 235.069,A -85,B 0,C 180,E1 19075.585,E2 19075.585} C_VEL
LIN {X 0,Y 402.636,Z 235.025,A -85,B 0,C 180,E1 19071.575,E2 19071.575} C_VEL
LIN {X 0,Y 402.642,Z 235.077,A -85,B 0,C 180,E1 19067.669,E2 19067.669} C_VEL
LIN {X 0,Y 402.678,Z 235.295,A -85,B 0,C 180,E1 19063.903,E2 19063.903} C_VEL
LIN {X 0,Y 403.932,Z 238.535,A -85,B 0,C 180,E1 19063.165,E2 19063.165} C_VEL
LIN {X 0,Y 405.243,Z 240.418,A -85,B 0,C 180,E1 19062.629,E2 19062.629} C_VEL
LIN {X 0,Y 407.271,Z 244.299,A -85,B 0,C 180,E1 19061.684,E2 19061.684} C_VEL
LIN {X 0,Y 413.414,Z 256.133,A -85,B 0,C 180,E1 19058.877,E2 19058.877} C_VEL
LIN {X 0,Y 419.642,Z 267.863,A -85,B 0,C 180,E1 19056.254,E2 19056.254} C_VEL
LIN {X 0,Y 428.362,Z 284.928,A -85,B 0,C 180,E1 19052.773,E2 19052.773} C_VEL
LIN {X 0,Y 438.2,Z 304.91,A -85,B 0,C 180,E1 19049.109,E2 19049.109} C_VEL
LIN {X 0,Y 447.883,Z 325.197,A -85,B 0,C 180,E1 19045.765,E2 19045.765} C_VEL
LIN {X 0,Y 449.321,Z 327.855,A -85,B 0,C 180,E1 19045.407,E2 19045.407} C_VEL
LIN {X 0,Y 468.235,Z 357.336,A -85,B 0,C 180,E1 19042.564,E2 19042.564} C_VEL
LIN {X 0,Y 452.672,Z 602.957,A -85,B 0,C 180,E1 19037.828,E2 19037.828} C_VEL
LIN {X 0,Y 447.532,Z 693.393,A -85,B 0,C 180,E1 19036.053,E2 19036.053} C_VEL
LIN {X 0,Y 445.154,Z 717.934,A -85,B 0,C 180,E1 19035.362,E2 19035.362} C_VEL
LIN {X 0,Y 442.01,Z 743.924,A -85,B 0,C 180,E1 19034.388,E2 19034.388} C_VEL
LIN {X 0,Y 438.665,Z 767.287,A -85,B 0,C 180,E1 19033.277,E2 19033.277} C_VEL
LIN {X 0,Y 435.005,Z 789.351,A -85,B 0,C 180,E1 19031.981,E2 19031.981} C_VEL
LIN {X 0,Y 430.985,Z 811.601,A -85,B 0,C 180,E1 19030.429,E2 19030.429} C_VEL
LIN {X 0,Y 426.902,Z 832.266,A -85,B 0,C 180,E1 19028.709,E2 19028.709} C_VEL
LIN {X 0,Y 422.445,Z 853.607,A -85,B 0,C 180,E1 19026.617,E2 19026.617} C_VEL
LIN {X 0,Y 418.442,Z 872.322,A -85,B 0,C 180,E1 19024.472,E2 19024.472} C_VEL
LIN {X 0,Y 414.703,Z 889.344,A -85,B 0,C 180,E1 19022.189,E2 19022.189} C_VEL
LIN {X 0,Y 411.274,Z 905.352,A -85,B 0,C 180,E1 19019.733,E2 19019.733} C_VEL
LIN {X 0,Y 408.245,Z 919.956,A -85,B 0,C 180,E1 19017.101,E2 19017.101} C_VEL
LIN {X 0,Y 405.668,Z 933.438,A -85,B 0,C 180,E1 19014.307,E2 19014.307} C_VEL
LIN {X 0,Y 403.61,Z 945.51,A -85,B 0,C 180,E1 19011.331,E2 19011.331} C_VEL
LIN {X 0,Y 402.131,Z 956.233,A -85,B 0,C 180,E1 19008.224,E2 19008.224} C_VEL
LIN {X 0,Y 401.262,Z 964.473,A -85,B 0,C 180,E1 19005.316,E2 19005.316} C_VEL
LIN {X 0,Y 400.787,Z 971.664,A -85,B 0,C 180,E1 19002.243,E2 19002.243} C_VEL
LIN {X 0,Y 400.673,Z 977.063,A -85,B 0,C 180,E1 18999.19,E2 18999.19} C_VEL
LIN {X 0,Y 400.742,Z 980.667,A -85,B 0,C 180,E1 18996.447,E2 18996.447} C_VEL
LIN {X 0,Y 400.863,Z 983.322,A -85,B 0,C 180,E1 18993.289,E2 18993.289} C_VEL
LIN {X 0,Y 400.918,Z 984.21,A -85,B 0,C 180,E1 18990.429,E2 18990.429} C_VEL
LIN {X 0,Y 400.889,Z 983.899,A -85,B 0,C 180,E1 18987.856,E2 18987.856} C_VEL
LIN {X 0,Y 400.745,Z 982.323,A -85,B 0,C 180,E1 18984.99,E2 18984.99} C_VEL
LIN {X 0,Y 400.626,Z 979.002,A -85,B 0,C 180,E1 18981.821,E2 18981.821} C_VEL
LIN {X 0,Y 400.627,Z 974.586,A -85,B 0,C 180,E1 18978.92,E2 18978.92} C_VEL
LIN {X 0,Y 400.962,Z 968.262,A -85,B 0,C 180,E1 18975.707,E2 18975.707} C_VEL
LIN {X 0,Y 401.793,Z 960.095,A -85,B 0,C 180,E1 18972.475,E2 18972.475} C_VEL
LIN {X 0,Y 403.174,Z 950.792,A -85,B 0,C 180,E1 18969.38,E2 18969.38} C_VEL
LIN {X 0,Y 405.368,Z 939.105,A -85,B 0,C 180,E1 18966.138,E2 18966.138} C_VEL
LIN {X 0,Y 408.289,Z 926.172,A -85,B 0,C 180,E1 18963.054,E2 18963.054} C_VEL
LIN {X 0,Y 412.067,Z 911.092,A -85,B 0,C 180,E1 18960.009,E2 18960.009} C_VEL
LIN {X 0,Y 416.581,Z 894.718,A -85,B 0,C 180,E1 18957.149,E2 18957.149} C_VEL
LIN {X 0,Y 421.538,Z 877.5,A -85,B 0,C 180,E1 18954.566,E2 18954.566} C_VEL
LIN {X 0,Y 427.349,Z 857.778,A -85,B 0,C 180,E1 18952.022,E2 18952.022} C_VEL
LIN {X 0,Y 433.471,Z 837.335,A -85,B 0,C 180,E1 18949.768,E2 18949.768} C_VEL
LIN {X 0,Y 439.677,Z 816.077,A -85,B 0,C 180,E1 18947.777,E2 18947.777} C_VEL
LIN {X 0,Y 446.355,Z 792.602,A -85,B 0,C 180,E1 18945.928,E2 18945.928} C_VEL
LIN {X 0,Y 452.978,Z 768.224,A -85,B 0,C 180,E1 18944.341,E2 18944.341} C_VEL
LIN {X 0,Y 459.135,Z 744.038,A -85,B 0,C 180,E1 18943.06,E2 18943.06} C_VEL
LIN {X 0,Y 464.777,Z 719.677,A -85,B 0,C 180,E1 18942.034,E2 18942.034} C_VEL
LIN {X 0,Y 469.696,Z 695.435,A -85,B 0,C 180,E1 18941.247,E2 18941.247} C_VEL
LIN {X 0,Y 483.334,Z 618.38,A -85,B 0,C 180,E1 18939.329,E2 18939.329} C_VEL
LIN {X 0,Y 493.481,Z 571.567,A -85,B 0,C 180,E1 18938.158,E2 18938.158} C_VEL
LIN {X 0,Y 469.597,Z 672.835,A -85,B 0,C 180,E1 18935.083,E2 18935.083} C_VEL
LIN {X 0,Y 463.135,Z 699.906,A -85,B 0,C 180,E1 18934.148,E2 18934.148} C_VEL
LIN {X 0,Y 456.993,Z 722.138,A -85,B 0,C 180,E1 18933.161,E2 18933.161} C_VEL
LIN {X 0,Y 450.356,Z 744.439,A -85,B 0,C 180,E1 18931.898,E2 18931.898} C_VEL
LIN {X 0,Y 443.484,Z 766.764,A -85,B 0,C 180,E1 18930.334,E2 18930.334} C_VEL
LIN {X 0,Y 436.829,Z 788.198,A -85,B 0,C 180,E1 18928.506,E2 18928.506} C_VEL
LIN {X 0,Y 430.938,Z 807.473,A -85,B 0,C 180,E1 18926.529,E2 18926.529} C_VEL
LIN {X 0,Y 425.668,Z 824.709,A -85,B 0,C 180,E1 18924.42,E2 18924.42} C_VEL
LIN {X 0,Y 420.984,Z 839.947,A -85,B 0,C 180,E1 18922.188,E2 18922.188} C_VEL
LIN {X 0,Y 416.975,Z 852.881,A -85,B 0,C 180,E1 18919.908,E2 18919.908} C_VEL
LIN {X 0,Y 413.753,Z 863.124,A -85,B 0,C 180,E1 18917.728,E2 18917.728} C_VEL
LIN {X 0,Y 410.689,Z 872.523,A -85,B 0,C 180,E1 18915.245,E2 18915.245} C_VEL
LIN {X 0,Y 408.052,Z 880.19,A -85,B 0,C 180,E1 18912.597,E2 18912.597} C_VEL
LIN {X 0,Y 405.987,Z 885.686,A -85,B 0,C 180,E1 18909.927,E2 18909.927} C_VEL
LIN {X 0,Y 404.518,Z 889.004,A -85,B 0,C 180,E1 18907.385,E2 18907.385} C_VEL
LIN {X 0,Y 403.429,Z 890.534,A -85,B 0,C 180,E1 18904.834,E2 18904.834} C_VEL
LIN {X 0,Y 402.684,Z 890.319,A -85,B 0,C 180,E1 18902.277,E2 18902.277} C_VEL
LIN {X 0,Y 402.235,Z 888.345,A -85,B 0,C 180,E1 18899.715,E2 18899.715} C_VEL
LIN {X 0,Y 402.024,Z 884.497,A -85,B 0,C 180,E1 18897.067,E2 18897.067} C_VEL
LIN {X 0,Y 402.075,Z 878.77,A -85,B 0,C 180,E1 18894.434,E2 18894.434} C_VEL
LIN {X 0,Y 402.387,Z 871.247,A -85,B 0,C 180,E1 18891.857,E2 18891.857} C_VEL
LIN {X 0,Y 402.97,Z 862.228,A -85,B 0,C 180,E1 18889.419,E2 18889.419} C_VEL
LIN {X 0,Y 403.897,Z 851.146,A -85,B 0,C 180,E1 18886.981,E2 18886.981} C_VEL
LIN {X 0,Y 405.115,Z 838.563,A -85,B 0,C 180,E1 18884.687,E2 18884.687} C_VEL
LIN {X 0,Y 406.656,Z 824.022,A -85,B 0,C 180,E1 18882.47,E2 18882.47} C_VEL
LIN {X 0,Y 408.451,Z 807.884,A -85,B 0,C 180,E1 18880.404,E2 18880.404} C_VEL
LIN {X 0,Y 410.452,Z 790.07,A -85,B 0,C 180,E1 18878.5,E2 18878.5} C_VEL
LIN {X 0,Y 412.515,Z 770.976,A -85,B 0,C 180,E1 18876.804,E2 18876.804} C_VEL
LIN {X 0,Y 414.606,Z 751.017,A -85,B 0,C 180,E1 18875.341,E2 18875.341} C_VEL
LIN {X 0,Y 416.732,Z 728.916,A -85,B 0,C 180,E1 18874.031,E2 18874.031} C_VEL
LIN {X 0,Y 418.597,Z 706.926,A -85,B 0,C 180,E1 18873.009,E2 18873.009} C_VEL
LIN {X 0,Y 420.286,Z 683.864,A -85,B 0,C 180,E1 18872.21,E2 18872.21} C_VEL
LIN {X 0,Y 430.531,Z 507.576,A -85,B 0,C 180,E1 18867.943,E2 18867.943} C_VEL
LIN {X 0,Y 425.719,Z 436.95,A -85,B 0,C 180,E1 18865.525,E2 18865.525} C_VEL
LIN {X 0,Y 432.556,Z 384.765,A -85,B 0,C 180,E1 18861.135,E2 18861.135} C_VEL
LIN {X 0,Y 434.747,Z 369.445,A -85,B 0,C 180,E1 18859.824,E2 18859.824} C_VEL
LIN {X 0,Y 436.878,Z 369.238,A -85,B 0,C 180,E1 18859.458,E2 18859.458} C_VEL
LIN {X 0,Y 440.571,Z 366.73,A -85,B 0,C 180,E1 18859.012,E2 18859.012} C_VEL
LIN {X 0,Y 443.446,Z 363.976,A -85,B 0,C 180,E1 18858.735,E2 18858.735} C_VEL
LIN {X 0,Y 447.29,Z 362.213,A -85,B 0,C 180,E1 18858.228,E2 18858.228} C_VEL
LIN {X 0,Y 452.013,Z 358.506,A -85,B 0,C 180,E1 18857.741,E2 18857.741} C_VEL
LIN {X 0,Y 457.127,Z 355.759,A -85,B 0,C 180,E1 18857.136,E2 18857.136} C_VEL
LIN {X 0,Y 461.074,Z 352.937,A -85,B 0,C 180,E1 18856.742,E2 18856.742} C_VEL
LIN {X 0,Y 464.419,Z 351.348,A -85,B 0,C 180,E1 18856.358,E2 18856.358} C_VEL
LIN {X 0,Y 465.273,Z 353.834,A -85,B 0,C 180,E1 18856.041,E2 18856.041} C_VEL
LIN {X 0,Y 464.706,Z 374.053,A -85,B 0,C 180,E1 18854.63,E2 18854.63} C_VEL
LIN {X 0,Y 458.913,Z 400.652,A -85,B 0,C 180,E1 18853.665,E2 18853.665} C_VEL
LIN {X 0,Y 454.883,Z 482.443,A -85,B 0,C 180,E1 18852.294,E2 18852.294} C_VEL
LIN {X 0,Y 450.628,Z 543.813,A -85,B 0,C 180,E1 18851.056,E2 18851.056} C_VEL
LIN {X 0,Y 445.098,Z 608.261,A -85,B 0,C 180,E1 18849.533,E2 18849.533} C_VEL
LIN {X 0,Y 441.209,Z 653.482,A -85,B 0,C 180,E1 18848.272,E2 18848.272} C_VEL
LIN {X 0,Y 439.257,Z 678.779,A -85,B 0,C 180,E1 18847.392,E2 18847.392} C_VEL
LIN {X 0,Y 437.018,Z 699.883,A -85,B 0,C 180,E1 18846.422,E2 18846.422} C_VEL
LIN {X 0,Y 434.264,Z 720.371,A -85,B 0,C 180,E1 18845.239,E2 18845.239} C_VEL
LIN {X 0,Y 431.083,Z 740.248,A -85,B 0,C 180,E1 18843.826,E2 18843.826} C_VEL
LIN {X 0,Y 427.636,Z 759.025,A -85,B 0,C 180,E1 18842.216,E2 18842.216} C_VEL
LIN {X 0,Y 423.984,Z 776.893,A -85,B 0,C 180,E1 18840.389,E2 18840.389} C_VEL
LIN {X 0,Y 420.21,Z 793.987,A -85,B 0,C 180,E1 18838.307,E2 18838.307} C_VEL
LIN {X 0,Y 416.587,Z 809.547,A -85,B 0,C 180,E1 18836.055,E2 18836.055} C_VEL
LIN {X 0,Y 416.054,Z 811.677,A -85,B 0,C 180,E1 18835.707,E2 18835.707} C_VEL
LIN {X 0,Y 413.964,Z 816.792,A -85,B 0,C 180,E1 18834.942,E2 18834.942} C_VEL
LIN {X 0,Y 405.606,Z 829.339,A -85,B 0,C 180,E1 18833.087,E2 18833.087} C_VEL
LIN {X 0,Y 403.593,Z 833.764,A -85,B 0,C 180,E1 18832.231,E2 18832.231} C_VEL
LIN {X 0,Y 400.764,Z 845.186,A -85,B 0,C 180,E1 18829.532,E2 18829.532} C_VEL
LIN {X 0,Y 398.356,Z 855.299,A -85,B 0,C 180,E1 18826.627,E2 18826.627} C_VEL
LIN {X 0,Y 396.472,Z 863.836,A -85,B 0,C 180,E1 18823.565,E2 18823.565} C_VEL
LIN {X 0,Y 395.142,Z 870.452,A -85,B 0,C 180,E1 18820.498,E2 18820.498} C_VEL
LIN {X 0,Y 394.317,Z 875.294,A -85,B 0,C 180,E1 18817.431,E2 18817.431} C_VEL
LIN {X 0,Y 393.853,Z 878.467,A -85,B 0,C 180,E1 18814.368,E2 18814.368} C_VEL
LIN {X 0,Y 393.662,Z 880.005,A -85,B 0,C 180,E1 18811.456,E2 18811.456} C_VEL
LIN {X 0,Y 393.658,Z 880.02,A -85,B 0,C 180,E1 18808.545,E2 18808.545} C_VEL
LIN {X 0,Y 393.845,Z 878.542,A -85,B 0,C 180,E1 18805.632,E2 18805.632} C_VEL
LIN {X 0,Y 394.311,Z 875.372,A -85,B 0,C 180,E1 18802.524,E2 18802.524} C_VEL
LIN {X 0,Y 395.114,Z 870.659,A -85,B 0,C 180,E1 18799.502,E2 18799.502} C_VEL
LIN {X 0,Y 396.436,Z 864.108,A -85,B 0,C 180,E1 18796.434,E2 18796.434} C_VEL
LIN {X 0,Y 398.3,Z 855.618,A -85,B 0,C 180,E1 18793.37,E2 18793.37} C_VEL
LIN {X 0,Y 400.692,Z 845.567,A -85,B 0,C 180,E1 18790.465,E2 18790.465} C_VEL
LIN {X 0,Y 403.555,Z 834.031,A -85,B 0,C 180,E1 18787.723,E2 18787.723} C_VEL
LIN {X 0,Y 406.827,Z 821.049,A -85,B 0,C 180,E1 18785.148,E2 18785.148} C_VEL
LIN {X 0,Y 410.422,Z 806.621,A -85,B 0,C 180,E1 18782.741,E2 18782.741} C_VEL
LIN {X 0,Y 414.255,Z 790.673,A -85,B 0,C 180,E1 18780.502,E2 18780.502} C_VEL
LIN {X 0,Y 418.229,Z 773.076,A -85,B 0,C 180,E1 18778.427,E2 18778.427} C_VEL
LIN {X 0,Y 421.949,Z 755.104,A -85,B 0,C 180,E1 18776.649,E2 18776.649} C_VEL
LIN {X 0,Y 425.438,Z 736.261,A -85,B 0,C 180,E1 18775.09,E2 18775.09} C_VEL
LIN {X 0,Y 428.589,Z 716.572,A -85,B 0,C 180,E1 18773.743,E2 18773.743} C_VEL
LIN {X 0,Y 431.311,Z 695.996,A -85,B 0,C 180,E1 18772.599,E2 18772.599} C_VEL
LIN {X 0,Y 433.518,Z 674.401,A -85,B 0,C 180,E1 18771.657,E2 18771.657} C_VEL
LIN {X 0,Y 436.584,Z 635.577,A -85,B 0,C 180,E1 18770.417,E2 18770.417} C_VEL
LIN {X 0,Y 442.217,Z 574.88,A -85,B 0,C 180,E1 18768.854,E2 18768.854} C_VEL
LIN {X 0,Y 447.096,Z 514.41,A -85,B 0,C 180,E1 18767.521,E2 18767.521} C_VEL
LIN {X 0,Y 450.829,Z 453.05,A -85,B 0,C 180,E1 18766.383,E2 18766.383} C_VEL
LIN {X 0,Y 453.44,Z 401.597,A -85,B 0,C 180,E1 18765.519,E2 18765.519} C_VEL
LIN {X 0,Y 459.348,Z 375.023,A -85,B 0,C 180,E1 18764.53,E2 18764.53} C_VEL
LIN {X 0,Y 459.819,Z 357.957,A -85,B 0,C 180,E1 18763.32,E2 18763.32} C_VEL
LIN {X 0,Y 453.126,Z 339.263,A -85,B 0,C 180,E1 18760.781,E2 18760.781} C_VEL
LIN {X 0,Y 445.964,Z 321.559,A -85,B 0,C 180,E1 18758.067,E2 18758.067} C_VEL
LIN {X 0,Y 438.631,Z 305.81,A -85,B 0,C 180,E1 18755.381,E2 18755.381} C_VEL
LIN {X 0,Y 430.985,Z 291.238,A -85,B 0,C 180,E1 18752.564,E2 18752.564} C_VEL
LIN {X 0,Y 424.483,Z 279.873,A -85,B 0,C 180,E1 18750.115,E2 18750.115} C_VEL
LIN {X 0,Y 418.521,Z 270.199,A -85,B 0,C 180,E1 18747.767,E2 18747.767} C_VEL
LIN {X 0,Y 414.86,Z 264.72,A -85,B 0,C 180,E1 18746.287,E2 18746.287} C_VEL
LIN {X 0,Y 411.559,Z 259.659,A -85,B 0,C 180,E1 18744.854,E2 18744.854} C_VEL
LIN {X 0,Y 408.684,Z 255.692,A -85,B 0,C 180,E1 18743.618,E2 18743.618} C_VEL
LIN {X 0,Y 407.759,Z 254.125,A -85,B 0,C 180,E1 18743.177,E2 18743.177} C_VEL
LIN {X 0,Y 404.939,Z 250.788,A -85,B 0,C 180,E1 18741.93,E2 18741.93} C_VEL
LIN {X 0,Y 403.917,Z 248.503,A -85,B 0,C 180,E1 18741.34,E2 18741.34} C_VEL
LIN {X 0,Y 401.052,Z 245.867,A -85,B 0,C 180,E1 18740.048,E2 18740.048} C_VEL
LIN {X 0,Y 399.313,Z 242.292,A -85,B 0,C 180,E1 18738.997,E2 18738.997} C_VEL
LIN {X 0,Y 396.223,Z 239.78,A -85,B 0,C 180,E1 18737.476,E2 18737.476} C_VEL
LIN {X 0,Y 394.845,Z 236.765,A -85,B 0,C 180,E1 18736.504,E2 18736.504} C_VEL
LIN {X 0,Y 394.719,Z 236.027,A -85,B 0,C 180,E1 18736.331,E2 18736.331} C_VEL
LIN {X 0,Y 394.715,Z 236.003,A -85,B 0,C 180,E1 18732.434,E2 18732.434} C_VEL
LIN {X 0,Y 394.724,Z 236.047,A -85,B 0,C 180,E1 18728.449,E2 18728.449} C_VEL
LIN {X 0,Y 394.716,Z 236.016,A -85,B 0,C 180,E1 18724.504,E2 18724.504} C_VEL
LIN {X 0,Y 394.72,Z 236.009,A -85,B 0,C 180,E1 18720.581,E2 18720.581} C_VEL
LIN {X 0,Y 394.723,Z 236.06,A -85,B 0,C 180,E1 18716.515,E2 18716.515} C_VEL
LIN {X 0,Y 394.725,Z 235.999,A -85,B 0,C 180,E1 18712.431,E2 18712.431} C_VEL
LIN {X 0,Y 394.725,Z 236.06,A -85,B 0,C 180,E1 18708.456,E2 18708.456} C_VEL
LIN {X 0,Y 394.723,Z 236.223,A -85,B 0,C 180,E1 18705.439,E2 18705.439} C_VEL
LIN {X 0,Y 396.103,Z 239.627,A -85,B 0,C 180,E1 18704.63,E2 18704.63} C_VEL
LIN {X 0,Y 397.354,Z 241.451,A -85,B 0,C 180,E1 18704.081,E2 18704.081} C_VEL
LIN {X 0,Y 399.276,Z 245.225,A -85,B 0,C 180,E1 18703.112,E2 18703.112} C_VEL
LIN {X 0,Y 404.844,Z 255.697,A -85,B 0,C 180,E1 18700.523,E2 18700.523} C_VEL
LIN {X 0,Y 412.442,Z 270.324,A -85,B 0,C 180,E1 18697.177,E2 18697.177} C_VEL
LIN {X 0,Y 420.762,Z 286.51,A -85,B 0,C 180,E1 18693.768,E2 18693.768} C_VEL
LIN {X 0,Y 430.872,Z 306.895,A -85,B 0,C 180,E1 18689.917,E2 18689.917} C_VEL
LIN {X 0,Y 441.101,Z 328.179,A -85,B 0,C 180,E1 18686.342,E2 18686.342} C_VEL
LIN {X 0,Y 461.877,Z 360.637,A -85,B 0,C 180,E1 18683.137,E2 18683.137} C_VEL
LIN {X 0,Y 445.47,Z 611.489,A -85,B 0,C 180,E1 18678.218,E2 18678.218} C_VEL
LIN {X 0,Y 440.619,Z 693.447,A -85,B 0,C 180,E1 18676.572,E2 18676.572} C_VEL
LIN {X 0,Y 438.181,Z 717.872,A -85,B 0,C 180,E1 18675.871,E2 18675.871} C_VEL
LIN {X 0,Y 434.969,Z 743.728,A -85,B 0,C 180,E1 18674.888,E2 18674.888} C_VEL
LIN {X 0,Y 431.633,Z 766.481,A -85,B 0,C 180,E1 18673.794,E2 18673.794} C_VEL
LIN {X 0,Y 427.886,Z 788.627,A -85,B 0,C 180,E1 18672.48,E2 18672.48} C_VEL
LIN {X 0,Y 423.763,Z 810.906,A -85,B 0,C 180,E1 18670.908,E2 18670.908} C_VEL
LIN {X 0,Y 419.579,Z 831.575,A -85,B 0,C 180,E1 18669.162,E2 18669.162} C_VEL
LIN {X 0,Y 415.003,Z 852.964,A -85,B 0,C 180,E1 18667.038,E2 18667.038} C_VEL
LIN {X 0,Y 410.924,Z 871.57,A -85,B 0,C 180,E1 18664.877,E2 18664.877} C_VEL
LIN {X 0,Y 406.955,Z 889.233,A -85,B 0,C 180,E1 18662.47,E2 18662.47} C_VEL
LIN {X 0,Y 403.342,Z 905.635,A -85,B 0,C 180,E1 18659.886,E2 18659.886} C_VEL
LIN {X 0,Y 400.265,Z 920.149,A -85,B 0,C 180,E1 18657.203,E2 18657.203} C_VEL
LIN {X 0,Y 397.541,Z 934.122,A -85,B 0,C 180,E1 18654.203,E2 18654.203} C_VEL
LIN {X 0,Y 395.598,Z 945.41,A -85,B 0,C 180,E1 18651.344,E2 18651.344} C_VEL
LIN {X 0,Y 394.063,Z 956.397,A -85,B 0,C 180,E1 18648.033,E2 18648.033} C_VEL
LIN {X 0,Y 393.258,Z 964.212,A -85,B 0,C 180,E1 18645.182,E2 18645.182} C_VEL
LIN {X 0,Y 392.785,Z 971.796,A -85,B 0,C 180,E1 18641.75,E2 18641.75} C_VEL
LIN {X 0,Y 392.716,Z 976.546,A -85,B 0,C 180,E1 18638.927,E2 18638.927} C_VEL
LIN {X 0,Y 392.812,Z 980.195,A -85,B 0,C 180,E1 18635.99,E2 18635.99} C_VEL
LIN {X 0,Y 392.931,Z 982.478,A -85,B 0,C 180,E1 18632.917,E2 18632.917} C_VEL
LIN {X 0,Y 392.993,Z 983.233,A -85,B 0,C 180,E1 18630.146,E2 18630.146} C_VEL
LIN {X 0,Y 392.923,Z 982.838,A -85,B 0,C 180,E1 18627.52,E2 18627.52} C_VEL
LIN {X 0,Y 392.774,Z 981.073,A -85,B 0,C 180,E1 18624.449,E2 18624.449} C_VEL
LIN {X 0,Y 392.632,Z 977.508,A -85,B 0,C 180,E1 18621.211,E2 18621.211} C_VEL
LIN {X 0,Y 392.68,Z 972.943,A -85,B 0,C 180,E1 18618.246,E2 18618.246} C_VEL
LIN {X 0,Y 393.149,Z 966.031,A -85,B 0,C 180,E1 18614.814,E2 18614.814} C_VEL
LIN {X 0,Y 394.093,Z 958.065,A -85,B 0,C 180,E1 18611.662,E2 18611.662} C_VEL
LIN {X 0,Y 395.854,Z 947.573,A -85,B 0,C 180,E1 18608.204,E2 18608.204} C_VEL
LIN {X 0,Y 398.258,Z 936.146,A -85,B 0,C 180,E1 18605.052,E2 18605.052} C_VEL
LIN {X 0,Y 401.89,Z 921.536,A -85,B 0,C 180,E1 18601.627,E2 18601.627} C_VEL
LIN {X 0,Y 405.979,Z 906.89,A -85,B 0,C 180,E1 18598.689,E2 18598.689} C_VEL
LIN {X 0,Y 410.944,Z 890.086,A -85,B 0,C 180,E1 18595.802,E2 18595.802} C_VEL
LIN {X 0,Y 416.595,Z 872.055,A -85,B 0,C 180,E1 18593.127,E2 18593.127} C_VEL
LIN {X 0,Y 422.605,Z 853.132,A -85,B 0,C 180,E1 18590.735,E2 18590.735} C_VEL
LIN {X 0,Y 429.388,Z 831.772,A -85,B 0,C 180,E1 18588.42,E2 18588.42} C_VEL
LIN {X 0,Y 436.361,Z 809.637,A -85,B 0,C 180,E1 18586.392,E2 18586.392} C_VEL
LIN {X 0,Y 443.373,Z 786.731,A -85,B 0,C 180,E1 18584.642,E2 18584.642} C_VEL
LIN {X 0,Y 450.057,Z 763.599,A -85,B 0,C 180,E1 18583.18,E2 18583.18} C_VEL
LIN {X 0,Y 456.498,Z 739.939,A -85,B 0,C 180,E1 18581.959,E2 18581.959} C_VEL
LIN {X 0,Y 462.208,Z 717.359,A -85,B 0,C 180,E1 18581.023,E2 18581.023} C_VEL
LIN {X 0,Y 467.629,Z 692.711,A -85,B 0,C 180,E1 18580.234,E2 18580.234} C_VEL
LIN {X 0,Y 481.28,Z 623.062,A -85,B 0,C 180,E1 18578.489,E2 18578.489} C_VEL
LIN {X 0,Y 484.763,Z 607.39,A -85,B 0,C 180,E1 18578.084,E2 18578.084} C_VEL
LIN {X 0,Y 463.628,Z 693.211,A -85,B 0,C 180,E1 18575.404,E2 18575.404} C_VEL
LIN {X 0,Y 456.879,Z 716.529,A -85,B 0,C 180,E1 18574.453,E2 18574.453} C_VEL
LIN {X 0,Y 449.865,Z 738.42,A -85,B 0,C 180,E1 18573.298,E2 18573.298} C_VEL
LIN {X 0,Y 442.192,Z 761.052,A -85,B 0,C 180,E1 18571.794,E2 18571.794} C_VEL
LIN {X 0,Y 434.461,Z 783.348,A -85,B 0,C 180,E1 18569.961,E2 18569.961} C_VEL
LIN {X 0,Y 427.57,Z 803.392,A -85,B 0,C 180,E1 18567.962,E2 18567.962} C_VEL
LIN {X 0,Y 421.307,Z 821.917,A -85,B 0,C 180,E1 18565.742,E2 18565.742} C_VEL
LIN {X 0,Y 416.071,Z 837.49,A -85,B 0,C 180,E1 18563.511,E2 18563.511} C_VEL
LIN {X 0,Y 411.566,Z 850.821,A -85,B 0,C 180,E1 18561.223,E2 18561.223} C_VEL
LIN {X 0,Y 407.505,Z 862.67,A -85,B 0,C 180,E1 18558.75,E2 18558.75} C_VEL
LIN {X 0,Y 404.257,Z 871.817,A -85,B 0,C 180,E1 18556.378,E2 18556.378} C_VEL
LIN {X 0,Y 401.41,Z 879.548,A -85,B 0,C 180,E1 18553.835,E2 18553.835} C_VEL
LIN {X 0,Y 399.007,Z 885.589,A -85,B 0,C 180,E1 18551.126,E2 18551.126} C_VEL
LIN {X 0,Y 397.256,Z 889.417,A -85,B 0,C 180,E1 18548.54,E2 18548.54} C_VEL
LIN {X 0,Y 396.023,Z 891.442,A -85,B 0,C 180,E1 18546.087,E2 18546.087} C_VEL
LIN {X 0,Y 395.082,Z 891.845,A -85,B 0,C 180,E1 18543.482,E2 18543.482} C_VEL
LIN {X 0,Y 394.473,Z 890.47,A -85,B 0,C 180,E1 18540.871,E2 18540.871} C_VEL
LIN {X 0,Y 394.138,Z 887.359,A -85,B 0,C 180,E1 18538.255,E2 18538.255} C_VEL
LIN {X 0,Y 394.06,Z 882.487,A -85,B 0,C 180,E1 18535.634,E2 18535.634} C_VEL
LIN {X 0,Y 394.256,Z 875.77,A -85,B 0,C 180,E1 18533.008,E2 18533.008} C_VEL
LIN {X 0,Y 394.704,Z 867.579,A -85,B 0,C 180,E1 18530.522,E2 18530.522} C_VEL
LIN {X 0,Y 395.478,Z 857.425,A -85,B 0,C 180,E1 18528.034,E2 18528.034} C_VEL
LIN {X 0,Y 396.553,Z 845.844,A -85,B 0,C 180,E1 18525.694,E2 18525.694} C_VEL
LIN {X 0,Y 397.993,Z 831.999,A -85,B 0,C 180,E1 18523.357,E2 18523.357} C_VEL
LIN {X 0,Y 399.72,Z 816.558,A -85,B 0,C 180,E1 18521.174,E2 18521.174} C_VEL
LIN {X 0,Y 401.687,Z 799.484,A -85,B 0,C 180,E1 18519.148,E2 18519.148} C_VEL
LIN {X 0,Y 403.836,Z 780.552,A -85,B 0,C 180,E1 18517.278,E2 18517.278} C_VEL
LIN {X 0,Y 405.964,Z 761.165,A -85,B 0,C 180,E1 18515.688,E2 18515.688} C_VEL
LIN {X 0,Y 408.237,Z 739.392,A -85,B 0,C 180,E1 18514.231,E2 18514.231} C_VEL
LIN {X 0,Y 410.237,Z 717.786,A -85,B 0,C 180,E1 18513.08,E2 18513.08} C_VEL
LIN {X 0,Y 412.11,Z 694.835,A -85,B 0,C 180,E1 18512.142,E2 18512.142} C_VEL
LIN {X 0,Y 413.709,Z 669.985,A -85,B 0,C 180,E1 18511.424,E2 18511.424} C_VEL
LIN {X 0,Y 423.42,Z 508.339,A -85,B 0,C 180,E1 18507.455,E2 18507.455} C_VEL
LIN {X 0,Y 418.715,Z 436.254,A -85,B 0,C 180,E1 18504.934,E2 18504.934} C_VEL
LIN {X 0,Y 425.681,Z 384.922,A -85,B 0,C 180,E1 18500.56,E2 18500.56} C_VEL
LIN {X 0,Y 426.131,Z 382.75,A -85,B 0,C 180,E1 18500.34,E2 18500.34} C_VEL
LIN {X 0,Y 427.915,Z 382.591,A -85,B 0,C 180,E1 18500.015,E2 18500.015} C_VEL
LIN {X 0,Y 431.503,Z 380.197,A -85,B 0,C 180,E1 18499.547,E2 18499.547} C_VEL
LIN {X 0,Y 434.781,Z 376.908,A -85,B 0,C 180,E1 18499.222,E2 18499.222} C_VEL
LIN {X 0,Y 438.189,Z 375.386,A -85,B 0,C 180,E1 18498.741,E2 18498.741} C_VEL
LIN {X 0,Y 442.82,Z 371.714,A -85,B 0,C 180,E1 18498.232,E2 18498.232} C_VEL
LIN {X 0,Y 444.353,Z 370.603,A -85,B 0,C 180,E1 18498.063,E2 18498.063} C_VEL
LIN {X 0,Y 449.493,Z 367.543,A -85,B 0,C 180,E1 18497.449,E2 18497.449} C_VEL
LIN {X 0,Y 452.639,Z 365.106,A -85,B 0,C 180,E1 18497.126,E2 18497.126} C_VEL
LIN {X 0,Y 458.648,Z 361.576,A -85,B 0,C 180,E1 18496.456,E2 18496.456} C_VEL
LIN {X 0,Y 459.587,Z 361.052,A -85,B 0,C 180,E1 18496.352,E2 18496.352} C_VEL
LIN {X 0,Y 459.113,Z 375.887,A -85,B 0,C 180,E1 18495.323,E2 18495.323} C_VEL
LIN {X 0,Y 453.096,Z 403.543,A -85,B 0,C 180,E1 18494.328,E2 18494.328} C_VEL
LIN {X 0,Y 448.959,Z 484.898,A -85,B 0,C 180,E1 18492.953,E2 18492.953} C_VEL
LIN {X 0,Y 444.604,Z 545.798,A -85,B 0,C 180,E1 18491.711,E2 18491.711} C_VEL
LIN {X 0,Y 438.973,Z 609.349,A -85,B 0,C 180,E1 18490.19,E2 18490.19} C_VEL
LIN {X 0,Y 434.943,Z 654.494,A -85,B 0,C 180,E1 18488.91,E2 18488.91} C_VEL
LIN {X 0,Y 432.878,Z 680.322,A -85,B 0,C 180,E1 18488,E2 18488} C_VEL
LIN {X 0,Y 430.481,Z 702.025,A -85,B 0,C 180,E1 18486.984,E2 18486.984} C_VEL
LIN {X 0,Y 427.457,Z 723.411,A -85,B 0,C 180,E1 18485.714,E2 18485.714} C_VEL
LIN {X 0,Y 424.019,Z 743.836,A -85,B 0,C 180,E1 18484.211,E2 18484.211} C_VEL
LIN {X 0,Y 420.34,Z 762.822,A -85,B 0,C 180,E1 18482.521,E2 18482.521} C_VEL
LIN {X 0,Y 416.453,Z 780.856,A -85,B 0,C 180,E1 18480.598,E2 18480.598} C_VEL
LIN {X 0,Y 412.647,Z 797.284,A -85,B 0,C 180,E1 18478.513,E2 18478.513} C_VEL
LIN {X 0,Y 408.993,Z 812.278,A -85,B 0,C 180,E1 18476.264,E2 18476.264} C_VEL
LIN {X 0,Y 405.404,Z 826.606,A -85,B 0,C 180,E1 18473.705,E2 18473.705} C_VEL
LIN {X 0,Y 403.593,Z 833.764,A -85,B 0,C 180,E1 18472.231,E2 18472.231} C_VEL
LIN {X 0,Y 401.613,Z 838.098,A -85,B 0,C 180,E1 18471.35,E2 18471.35} C_VEL
LIN {X 0,Y 393.52,Z 848.674,A -85,B 0,C 180,E1 18469.18,E2 18469.18} C_VEL
LIN {X 0,Y 391.69,Z 852.277,A -85,B 0,C 180,E1 18468.212,E2 18468.212} C_VEL
LIN {X 0,Y 389.483,Z 861.436,A -85,B 0,C 180,E1 18465.18,E2 18465.18} C_VEL
LIN {X 0,Y 387.84,Z 868.881,A -85,B 0,C 180,E1 18462.054,E2 18462.054} C_VEL
LIN {X 0,Y 386.745,Z 874.456,A -85,B 0,C 180,E1 18458.924,E2 18458.924} C_VEL
LIN {X 0,Y 386.124,Z 878.167,A -85,B 0,C 180,E1 18455.946,E2 18455.946} C_VEL
LIN {X 0,Y 385.79,Z 880.481,A -85,B 0,C 180,E1 18452.823,E2 18452.823} C_VEL
LIN {X 0,Y 385.713,Z 881.216,A -85,B 0,C 180,E1 18449.852,E2 18449.852} C_VEL
LIN {X 0,Y 385.816,Z 880.333,A -85,B 0,C 180,E1 18446.732,E2 18446.732} C_VEL
LIN {X 0,Y 386.158,Z 877.967,A -85,B 0,C 180,E1 18443.757,E2 18443.757} C_VEL
LIN {X 0,Y 386.888,Z 873.665,A -85,B 0,C 180,E1 18440.479,E2 18440.479} C_VEL
LIN {X 0,Y 388.069,Z 867.79,A -85,B 0,C 180,E1 18437.349,E2 18437.349} C_VEL
LIN {X 0,Y 389.714,Z 860.493,A -85,B 0,C 180,E1 18434.372,E2 18434.372} C_VEL
LIN {X 0,Y 391.951,Z 851.375,A -85,B 0,C 180,E1 18431.405,E2 18431.405} C_VEL
LIN {X 0,Y 394.838,Z 840.203,A -85,B 0,C 180,E1 18428.457,E2 18428.457} C_VEL
LIN {X 0,Y 398.208,Z 827.425,A -85,B 0,C 180,E1 18425.682,E2 18425.682} C_VEL
LIN {X 0,Y 401.975,Z 813.051,A -85,B 0,C 180,E1 18423.082,E2 18423.082} C_VEL
LIN {X 0,Y 405.796,Z 798.001,A -85,B 0,C 180,E1 18420.799,E2 18420.799} C_VEL
LIN {X 0,Y 409.769,Z 781.494,A -85,B 0,C 180,E1 18418.685,E2 18418.685} C_VEL
LIN {X 0,Y 413.668,Z 764.057,A -85,B 0,C 180,E1 18416.806,E2 18416.806} C_VEL
LIN {X 0,Y 417.35,Z 745.801,A -85,B 0,C 180,E1 18415.152,E2 18415.152} C_VEL
LIN {X 0,Y 420.859,Z 725.832,A -85,B 0,C 180,E1 18413.65,E2 18413.65} C_VEL
LIN {X 0,Y 424.008,Z 704.553,A -85,B 0,C 180,E1 18412.355,E2 18412.355} C_VEL
LIN {X 0,Y 426.552,Z 682.574,A -85,B 0,C 180,E1 18411.3,E2 18411.3} C_VEL
LIN {X 0,Y 428.685,Z 657.213,A -85,B 0,C 180,E1 18410.384,E2 18410.384} C_VEL
LIN {X 0,Y 432.655,Z 613.761,A -85,B 0,C 180,E1 18409.118,E2 18409.118} C_VEL
LIN {X 0,Y 438.249,Z 553.448,A -85,B 0,C 180,E1 18407.641,E2 18407.641} C_VEL
LIN {X 0,Y 442.721,Z 494.691,A -85,B 0,C 180,E1 18406.408,E2 18406.408} C_VEL
LIN {X 0,Y 446.474,Z 426.656,A -85,B 0,C 180,E1 18405.222,E2 18405.222} C_VEL
LIN {X 0,Y 447.695,Z 404.406,A -85,B 0,C 180,E1 18404.837,E2 18404.837} C_VEL
LIN {X 0,Y 453.87,Z 376.827,A -85,B 0,C 180,E1 18403.822,E2 18403.822} C_VEL
LIN {X 0,Y 454.278,Z 362.011,A -85,B 0,C 180,E1 18402.768,E2 18402.768} C_VEL
LIN {X 0,Y 447.684,Z 343.432,A -85,B 0,C 180,E1 18400.195,E2 18400.195} C_VEL
LIN {X 0,Y 440.52,Z 325.873,A -85,B 0,C 180,E1 18397.467,E2 18397.467} C_VEL
LIN {X 0,Y 434.093,Z 311.731,A -85,B 0,C 180,E1 18394.998,E2 18394.998} C_VEL
LIN {X 0,Y 426.278,Z 296.51,A -85,B 0,C 180,E1 18392.013,E2 18392.013} C_VEL
LIN {X 0,Y 419.921,Z 285.436,A -85,B 0,C 180,E1 18389.531,E2 18389.531} C_VEL
LIN {X 0,Y 414.738,Z 276.821,A -85,B 0,C 180,E1 18387.418,E2 18387.418} C_VEL
LIN {X 0,Y 411.157,Z 271.383,A -85,B 0,C 180,E1 18385.921,E2 18385.921} C_VEL
LIN {X 0,Y 407.9,Z 266.38,A -85,B 0,C 180,E1 18384.474,E2 18384.474} C_VEL
LIN {X 0,Y 405.036,Z 262.018,A -85,B 0,C 180,E1 18383.15,E2 18383.15} C_VEL
LIN {X 0,Y 401.5,Z 257.301,A -85,B 0,C 180,E1 18381.475,E2 18381.475} C_VEL
LIN {X 0,Y 400.444,Z 255.504,A -85,B 0,C 180,E1 18380.92,E2 18380.92} C_VEL
LIN {X 0,Y 397.56,Z 252.262,A -85,B 0,C 180,E1 18379.504,E2 18379.504} C_VEL
LIN {X 0,Y 396.257,Z 249.595,A -85,B 0,C 180,E1 18378.691,E2 18378.691} C_VEL
LIN {X 0,Y 393.207,Z 246.736,A -85,B 0,C 180,E1 18377.08,E2 18377.08} C_VEL
LIN {X 0,Y 391.725,Z 243.456,A -85,B 0,C 180,E1 18376.002,E2 18376.002} C_VEL
LIN {X 0,Y 388.66,Z 241.248,A -85,B 0,C 180,E1 18374.223,E2 18374.223} C_VEL
LIN {X 0,Y 387.021,Z 238.188,A -85,B 0,C 180,E1 18372.875,E2 18372.875} C_VEL
LIN {X 0,Y 386.776,Z 236.99,A -85,B 0,C 180,E1 18372.466,E2 18372.466} C_VEL
LIN {X 0,Y 386.785,Z 237.035,A -85,B 0,C 180,E1 18368.474,E2 18368.474} C_VEL
LIN {X 0,Y 386.777,Z 237.005,A -85,B 0,C 180,E1 18364.448,E2 18364.448} C_VEL
LIN {X 0,Y 386.783,Z 236.994,A -85,B 0,C 180,E1 18360.444,E2 18360.444} C_VEL
LIN {X 0,Y 386.784,Z 237.05,A -85,B 0,C 180,E1 18356.443,E2 18356.443} C_VEL
LIN {X 0,Y 386.786,Z 236.986,A -85,B 0,C 180,E1 18352.424,E2 18352.424} C_VEL
LIN {X 0,Y 386.785,Z 237.049,A -85,B 0,C 180,E1 18348.367,E2 18348.367} C_VEL
LIN {X 0,Y 386.804,Z 237.252,A -85,B 0,C 180,E1 18347.003,E2 18347.003} C_VEL
LIN {X 0,Y 388.187,Z 240.679,A -85,B 0,C 180,E1 18346.14,E2 18346.14} C_VEL
LIN {X 0,Y 389.427,Z 242.534,A -85,B 0,C 180,E1 18345.578,E2 18345.578} C_VEL
LIN {X 0,Y 391.397,Z 246.244,A -85,B 0,C 180,E1 18344.592,E2 18344.592} C_VEL
LIN {X 0,Y 395.007,Z 253.287,A -85,B 0,C 180,E1 18342.773,E2 18342.773} C_VEL
LIN {X 0,Y 399.489,Z 261.557,A -85,B 0,C 180,E1 18340.708,E2 18340.708} C_VEL
LIN {X 0,Y 406.761,Z 275.608,A -85,B 0,C 180,E1 18337.451,E2 18337.451} C_VEL
LIN {X 0,Y 414.763,Z 291.217,A -85,B 0,C 180,E1 18334.129,E2 18334.129} C_VEL
LIN {X 0,Y 424.484,Z 311.003,A -85,B 0,C 180,E1 18330.352,E2 18330.352} C_VEL
LIN {X 0,Y 433.421,Z 329.484,A -85,B 0,C 180,E1 18327.21,E2 18327.21} C_VEL
LIN {X 0,Y 452.32,Z 358.906,A -85,B 0,C 180,E1 18324.199,E2 18324.199} C_VEL
LIN {X 0,Y 455.523,Z 364.299,A -85,B 0,C 180,E1 18323.71,E2 18323.71} C_VEL
LIN {X 0,Y 438.872,Z 609.311,A -85,B 0,C 180,E1 18318.824,E2 18318.824} C_VEL
LIN {X 0,Y 433.695,Z 693.457,A -85,B 0,C 180,E1 18317.098,E2 18317.098} C_VEL
LIN {X 0,Y 431.196,Z 717.825,A -85,B 0,C 180,E1 18316.386,E2 18316.386} C_VEL
LIN {X 0,Y 427.945,Z 743.337,A -85,B 0,C 180,E1 18315.402,E2 18315.402} C_VEL
LIN {X 0,Y 424.437,Z 766.658,A -85,B 0,C 180,E1 18314.261,E2 18314.261} C_VEL
LIN {X 0,Y 420.604,Z 788.712,A -85,B 0,C 180,E1 18312.929,E2 18312.929} C_VEL
LIN {X 0,Y 416.379,Z 810.971,A -85,B 0,C 180,E1 18311.329,E2 18311.329} C_VEL
LIN {X 0,Y 412.115,Z 831.579,A -85,B 0,C 180,E1 18309.56,E2 18309.56} C_VEL
LIN {X 0,Y 407.434,Z 852.923,A -85,B 0,C 180,E1 18307.401,E2 18307.401} C_VEL
LIN {X 0,Y 403.261,Z 871.48,A -85,B 0,C 180,E1 18305.204,E2 18305.204} C_VEL
LIN {X 0,Y 399.203,Z 889.058,A -85,B 0,C 180,E1 18302.753,E2 18302.753} C_VEL
LIN {X 0,Y 395.414,Z 905.839,A -85,B 0,C 180,E1 18300.045,E2 18300.045} C_VEL
LIN {X 0,Y 392.287,Z 920.306,A -85,B 0,C 180,E1 18297.309,E2 18297.309} C_VEL
LIN {X 0,Y 389.531,Z 934.128,A -85,B 0,C 180,E1 18294.249,E2 18294.249} C_VEL
LIN {X 0,Y 387.573,Z 945.334,A -85,B 0,C 180,E1 18291.331,E2 18291.331} C_VEL
LIN {X 0,Y 386.099,Z 955.744,A -85,B 0,C 180,E1 18288.105,E2 18288.105} C_VEL
LIN {X 0,Y 385.254,Z 963.925,A -85,B 0,C 180,E1 18285.043,E2 18285.043} C_VEL
LIN {X 0,Y 384.815,Z 971.245,A -85,B 0,C 180,E1 18281.596,E2 18281.596} C_VEL
LIN {X 0,Y 384.768,Z 975.767,A -85,B 0,C 180,E1 18278.819,E2 18278.819} C_VEL
LIN {X 0,Y 384.887,Z 979.537,A -85,B 0,C 180,E1 18275.665,E2 18275.665} C_VEL
LIN {X 0,Y 385.007,Z 981.616,A -85,B 0,C 180,E1 18272.53,E2 18272.53} C_VEL
LIN {X 0,Y 385.054,Z 982.237,A -85,B 0,C 180,E1 18269.851,E2 18269.851} C_VEL
LIN {X 0,Y 384.962,Z 981.766,A -85,B 0,C 180,E1 18267.171,E2 18267.171} C_VEL
LIN {X 0,Y 384.793,Z 979.889,A -85,B 0,C 180,E1 18264.034,E2 18264.034} C_VEL
LIN {X 0,Y 384.661,Z 976.212,A -85,B 0,C 180,E1 18260.725,E2 18260.725} C_VEL
LIN {X 0,Y 384.754,Z 971.3,A -85,B 0,C 180,E1 18257.543,E2 18257.543} C_VEL
LIN {X 0,Y 385.317,Z 964.153,A -85,B 0,C 180,E1 18254.034,E2 18254.034} C_VEL
LIN {X 0,Y 386.425,Z 956.056,A -85,B 0,C 180,E1 18250.814,E2 18250.814} C_VEL
LIN {X 0,Y 388.557,Z 944.759,A -85,B 0,C 180,E1 18247.111,E2 18247.111} C_VEL
LIN {X 0,Y 391.457,Z 932.66,A -85,B 0,C 180,E1 18243.775,E2 18243.775} C_VEL
LIN {X 0,Y 395.148,Z 919.02,A -85,B 0,C 180,E1 18240.6,E2 18240.6} C_VEL
LIN {X 0,Y 399.86,Z 903.525,A -85,B 0,C 180,E1 18237.477,E2 18237.477} C_VEL
LIN {X 0,Y 405.323,Z 886.524,A -85,B 0,C 180,E1 18234.569,E2 18234.569} C_VEL
LIN {X 0,Y 411.794,Z 867.242,A -85,B 0,C 180,E1 18231.744,E2 18231.744} C_VEL
LIN {X 0,Y 418.532,Z 847.682,A -85,B 0,C 180,E1 18229.292,E2 18229.292} C_VEL
LIN {X 0,Y 425.937,Z 826.015,A -85,B 0,C 180,E1 18227.004,E2 18227.004} C_VEL
LIN {X 0,Y 433.473,Z 803.573,A -85,B 0,C 180,E1 18225.008,E2 18225.008} C_VEL
LIN {X 0,Y 441.288,Z 779.648,A -85,B 0,C 180,E1 18223.242,E2 18223.242} C_VEL
LIN {X 0,Y 448.406,Z 756.913,A -85,B 0,C 180,E1 18221.86,E2 18221.86} C_VEL
LIN {X 0,Y 455.78,Z 731.482,A -85,B 0,C 180,E1 18220.619,E2 18220.619} C_VEL
LIN {X 0,Y 462.797,Z 704.676,A -85,B 0,C 180,E1 18219.625,E2 18219.625} C_VEL
LIN {X 0,Y 469.158,Z 676.067,A -85,B 0,C 180,E1 18218.834,E2 18218.834} C_VEL
LIN {X 0,Y 476.133,Z 643.016,A -85,B 0,C 180,E1 18218.005,E2 18218.005} C_VEL
LIN {X 0,Y 462.977,Z 693.676,A -85,B 0,C 180,E1 18216.407,E2 18216.407} C_VEL
LIN {X 0,Y 456.058,Z 715.992,A -85,B 0,C 180,E1 18215.521,E2 18215.521} C_VEL
LIN {X 0,Y 448.511,Z 737.483,A -85,B 0,C 180,E1 18214.412,E2 18214.412} C_VEL
LIN {X 0,Y 440.185,Z 759.718,A -85,B 0,C 180,E1 18212.959,E2 18212.959} C_VEL
LIN {X 0,Y 431.751,Z 781.709,A -85,B 0,C 180,E1 18211.172,E2 18211.172} C_VEL
LIN {X 0,Y 423.949,Z 802.145,A -85,B 0,C 180,E1 18209.146,E2 18209.146} C_VEL
LIN {X 0,Y 417.034,Z 820.526,A -85,B 0,C 180,E1 18206.946,E2 18206.946} C_VEL
LIN {X 0,Y 410.915,Z 836.989,A -85,B 0,C 180,E1 18204.589,E2 18204.589} C_VEL
LIN {X 0,Y 405.68,Z 851.086,A -85,B 0,C 180,E1 18202.154,E2 18202.154} C_VEL
LIN {X 0,Y 401.228,Z 862.95,A -85,B 0,C 180,E1 18199.66,E2 18199.66} C_VEL
LIN {X 0,Y 397.481,Z 872.726,A -85,B 0,C 180,E1 18197.117,E2 18197.117} C_VEL
LIN {X 0,Y 394.521,Z 880.094,A -85,B 0,C 180,E1 18194.681,E2 18194.681} C_VEL
LIN {X 0,Y 392.095,Z 885.785,A -85,B 0,C 180,E1 18192.22,E2 18192.22} C_VEL
LIN {X 0,Y 389.965,Z 890.185,A -85,B 0,C 180,E1 18189.445,E2 18189.445} C_VEL
LIN {X 0,Y 388.387,Z 892.589,A -85,B 0,C 180,E1 18186.653,E2 18186.653} C_VEL
LIN {X 0,Y 387.318,Z 893.073,A -85,B 0,C 180,E1 18183.997,E2 18183.997} C_VEL
LIN {X 0,Y 386.62,Z 891.814,A -85,B 0,C 180,E1 18181.334,E2 18181.334} C_VEL
LIN {X 0,Y 386.227,Z 888.84,A -85,B 0,C 180,E1 18178.665,E2 18178.665} C_VEL
LIN {X 0,Y 386.098,Z 884.094,A -85,B 0,C 180,E1 18175.99,E2 18175.99} C_VEL
LIN {X 0,Y 386.253,Z 877.511,A -85,B 0,C 180,E1 18173.31,E2 18173.31} C_VEL
LIN {X 0,Y 386.708,Z 868.943,A -85,B 0,C 180,E1 18170.625,E2 18170.625} C_VEL
LIN {X 0,Y 387.48,Z 858.836,A -85,B 0,C 180,E1 18168.086,E2 18168.086} C_VEL
LIN {X 0,Y 388.564,Z 847.335,A -85,B 0,C 180,E1 18165.698,E2 18165.698} C_VEL
LIN {X 0,Y 390.022,Z 833.555,A -85,B 0,C 180,E1 18163.314,E2 18163.314} C_VEL
LIN {X 0,Y 391.77,Z 818.194,A -85,B 0,C 180,E1 18161.087,E2 18161.087} C_VEL
LIN {X 0,Y 393.77,Z 801.231,A -85,B 0,C 180,E1 18159.02,E2 18159.02} C_VEL
LIN {X 0,Y 395.966,Z 782.544,A -85,B 0,C 180,E1 18157.115,E2 18157.115} C_VEL
LIN {X 0,Y 398.192,Z 762.729,A -85,B 0,C 180,E1 18155.444,E2 18155.444} C_VEL
LIN {X 0,Y 400.469,Z 741.56,A -85,B 0,C 180,E1 18153.983,E2 18153.983} C_VEL
LIN {X 0,Y 402.655,Z 718.86,A -85,B 0,C 180,E1 18152.732,E2 18152.732} C_VEL
LIN {X 0,Y 404.637,Z 695.56,A -85,B 0,C 180,E1 18151.747,E2 18151.747} C_VEL
LIN {X 0,Y 406.317,Z 670.767,A -85,B 0,C 180,E1 18151.001,E2 18151.001} C_VEL
LIN {X 0,Y 416.368,Z 509.241,A -85,B 0,C 180,E1 18146.95,E2 18146.95} C_VEL
LIN {X 0,Y 411.819,Z 434.892,A -85,B 0,C 180,E1 18144.272,E2 18144.272} C_VEL
LIN {X 0,Y 417.314,Z 396.542,A -85,B 0,C 180,E1 18140.924,E2 18140.924} C_VEL
LIN {X 0,Y 419.025,Z 396.405,A -85,B 0,C 180,E1 18140.599,E2 18140.599} C_VEL
LIN {X 0,Y 422.554,Z 393.983,A -85,B 0,C 180,E1 18140.113,E2 18140.113} C_VEL
LIN {X 0,Y 426.507,Z 390.073,A -85,B 0,C 180,E1 18139.68,E2 18139.68} C_VEL
LIN {X 0,Y 429.92,Z 388.343,A -85,B 0,C 180,E1 18139.191,E2 18139.191} C_VEL
LIN {X 0,Y 434.535,Z 384.439,A -85,B 0,C 180,E1 18138.669,E2 18138.669} C_VEL
LIN {X 0,Y 436.012,Z 383.401,A -85,B 0,C 180,E1 18138.49,E2 18138.49} C_VEL
LIN {X 0,Y 441.133,Z 380.207,A -85,B 0,C 180,E1 18137.861,E2 18137.861} C_VEL
LIN {X 0,Y 444.314,Z 377.511,A -85,B 0,C 180,E1 18137.536,E2 18137.536} C_VEL
LIN {X 0,Y 450.224,Z 373.917,A -85,B 0,C 180,E1 18136.84,E2 18136.84} C_VEL
LIN {X 0,Y 453.541,Z 371.552,A -85,B 0,C 180,E1 18136.496,E2 18136.496} C_VEL
LIN {X 0,Y 453.879,Z 371.446,A -85,B 0,C 180,E1 18136.451,E2 18136.451} C_VEL
LIN {X 0,Y 453.587,Z 377.698,A -85,B 0,C 180,E1 18136.033,E2 18136.033} C_VEL
LIN {X 0,Y 447.352,Z 406.224,A -85,B 0,C 180,E1 18135.011,E2 18135.011} C_VEL
LIN {X 0,Y 443.108,Z 487.162,A -85,B 0,C 180,E1 18133.633,E2 18133.633} C_VEL
LIN {X 0,Y 438.689,Z 547.175,A -85,B 0,C 180,E1 18132.397,E2 18132.397} C_VEL
LIN {X 0,Y 433.081,Z 608.665,A -85,B 0,C 180,E1 18130.912,E2 18130.912} C_VEL
LIN {X 0,Y 428.889,Z 653.731,A -85,B 0,C 180,E1 18129.626,E2 18129.626} C_VEL
LIN {X 0,Y 426.647,Z 680.87,A -85,B 0,C 180,E1 18128.667,E2 18128.667} C_VEL
LIN {X 0,Y 424.281,Z 701.902,A -85,B 0,C 180,E1 18127.683,E2 18127.683} C_VEL
LIN {X 0,Y 421.328,Z 722.527,A -85,B 0,C 180,E1 18126.468,E2 18126.468} C_VEL
LIN {X 0,Y 417.968,Z 742.211,A -85,B 0,C 180,E1 18125.04,E2 18125.04} C_VEL
LIN {X 0,Y 414.191,Z 761.378,A -85,B 0,C 180,E1 18123.355,E2 18123.355} C_VEL
LIN {X 0,Y 410.178,Z 779.564,A -85,B 0,C 180,E1 18121.439,E2 18121.439} C_VEL
LIN {X 0,Y 406.046,Z 796.826,A -85,B 0,C 180,E1 18119.262,E2 18119.262} C_VEL
LIN {X 0,Y 402.086,Z 812.466,A -85,B 0,C 180,E1 18116.91,E2 18116.91} C_VEL
LIN {X 0,Y 398.304,Z 826.924,A -85,B 0,C 180,E1 18114.312,E2 18114.312} C_VEL
LIN {X 0,Y 394.918,Z 839.765,A -85,B 0,C 180,E1 18111.538,E2 18111.538} C_VEL
LIN {X 0,Y 392.014,Z 851.002,A -85,B 0,C 180,E1 18108.592,E2 18108.592} C_VEL
LIN {X 0,Y 391.69,Z 852.277,A -85,B 0,C 180,E1 18108.212,E2 18108.212} C_VEL
LIN {X 0,Y 389.915,Z 855.755,A -85,B 0,C 180,E1 18107.223,E2 18107.223} C_VEL
LIN {X 0,Y 381.987,Z 864.585,A -85,B 0,C 180,E1 18104.609,E2 18104.609} C_VEL
LIN {X 0,Y 380.731,Z 866.883,A -85,B 0,C 180,E1 18103.688,E2 18103.688} C_VEL
LIN {X 0,Y 379.318,Z 873.312,A -85,B 0,C 180,E1 18100.48,E2 18100.48} C_VEL
LIN {X 0,Y 378.415,Z 878.087,A -85,B 0,C 180,E1 18097.134,E2 18097.134} C_VEL
LIN {X 0,Y 377.961,Z 880.797,A -85,B 0,C 180,E1 18094.096,E2 18094.096} C_VEL
LIN {X 0,Y 377.77,Z 882.092,A -85,B 0,C 180,E1 18090.91,E2 18090.91} C_VEL
LIN {X 0,Y 377.819,Z 881.851,A -85,B 0,C 180,E1 18087.877,E2 18087.877} C_VEL
LIN {X 0,Y 378.106,Z 880.012,A -85,B 0,C 180,E1 18084.689,E2 18084.689} C_VEL
LIN {X 0,Y 378.69,Z 876.473,A -85,B 0,C 180,E1 18081.497,E2 18081.497} C_VEL
LIN {X 0,Y 379.696,Z 871.459,A -85,B 0,C 180,E1 18078.415,E2 18078.415} C_VEL
LIN {X 0,Y 381.253,Z 864.611,A -85,B 0,C 180,E1 18075.262,E2 18075.262} C_VEL
LIN {X 0,Y 383.432,Z 855.952,A -85,B 0,C 180,E1 18072.144,E2 18072.144} C_VEL
LIN {X 0,Y 386.143,Z 845.81,A -85,B 0,C 180,E1 18069.194,E2 18069.194} C_VEL
LIN {X 0,Y 389.371,Z 834.087,A -85,B 0,C 180,E1 18066.384,E2 18066.384} C_VEL
LIN {X 0,Y 393.059,Z 820.771,A -85,B 0,C 180,E1 18063.728,E2 18063.728} C_VEL
LIN {X 0,Y 397.211,Z 805.365,A -85,B 0,C 180,E1 18061.166,E2 18061.166} C_VEL
LIN {X 0,Y 401.443,Z 788.927,A -85,B 0,C 180,E1 18058.88,E2 18058.88} C_VEL
LIN {X 0,Y 405.661,Z 771.278,A -85,B 0,C 180,E1 18056.825,E2 18056.825} C_VEL
LIN {X 0,Y 409.732,Z 752.541,A -85,B 0,C 180,E1 18055.007,E2 18055.007} C_VEL
LIN {X 0,Y 413.555,Z 732.404,A -85,B 0,C 180,E1 18053.39,E2 18053.39} C_VEL
LIN {X 0,Y 416.899,Z 711.64,A -85,B 0,C 180,E1 18052.034,E2 18052.034} C_VEL
LIN {X 0,Y 419.68,Z 689.938,A -85,B 0,C 180,E1 18050.904,E2 18050.904} C_VEL
LIN {X 0,Y 421.825,Z 667.382,A -85,B 0,C 180,E1 18050.009,E2 18050.009} C_VEL
LIN {X 0,Y 425.72,Z 623.989,A -85,B 0,C 180,E1 18048.673,E2 18048.673} C_VEL
LIN {X 0,Y 431.631,Z 563.511,A -85,B 0,C 180,E1 18047.136,E2 18047.136} C_VEL
LIN {X 0,Y 436.608,Z 501.534,A -85,B 0,C 180,E1 18045.801,E2 18045.801} C_VEL
LIN {X 0,Y 440.103,Z 442.423,A -85,B 0,C 180,E1 18044.74,E2 18044.74} C_VEL
LIN {X 0,Y 442.011,Z 407.151,A -85,B 0,C 180,E1 18044.138,E2 18044.138} C_VEL
LIN {X 0,Y 448.465,Z 378.513,A -85,B 0,C 180,E1 18043.088,E2 18043.088} C_VEL
LIN {X 0,Y 448.812,Z 366.097,A -85,B 0,C 180,E1 18042.199,E2 18042.199} C_VEL
LIN {X 0,Y 442.169,Z 347.278,A -85,B 0,C 180,E1 18039.546,E2 18039.546} C_VEL
LIN {X 0,Y 435.242,Z 330.249,A -85,B 0,C 180,E1 18036.842,E2 18036.842} C_VEL
LIN {X 0,Y 429.223,Z 316.975,A -85,B 0,C 180,E1 18034.477,E2 18034.477} C_VEL
LIN {X 0,Y 423.212,Z 305.007,A -85,B 0,C 180,E1 18032.113,E2 18032.113} C_VEL
LIN {X 0,Y 416.718,Z 293.035,A -85,B 0,C 180,E1 18029.465,E2 18029.465} C_VEL
LIN {X 0,Y 410.973,Z 283.436,A -85,B 0,C 180,E1 18027.063,E2 18027.063} C_VEL
LIN {X 0,Y 407.293,Z 277.723,A -85,B 0,C 180,E1 18025.444,E2 18025.444} C_VEL
LIN {X 0,Y 404.436,Z 273.266,A -85,B 0,C 180,E1 18024.153,E2 18024.153} C_VEL
LIN {X 0,Y 400.989,Z 268.067,A -85,B 0,C 180,E1 18022.505,E2 18022.505} C_VEL
LIN {X 0,Y 398.189,Z 264.051,A -85,B 0,C 180,E1 18021.083,E2 18021.083} C_VEL
LIN {X 0,Y 397.363,Z 262.698,A -85,B 0,C 180,E1 18020.627,E2 18020.627} C_VEL
LIN {X 0,Y 394.418,Z 259.15,A -85,B 0,C 180,E1 18019.127,E2 18019.127} C_VEL
LIN {X 0,Y 393.235,Z 256.865,A -85,B 0,C 180,E1 18018.379,E2 18018.379} C_VEL
LIN {X 0,Y 390.311,Z 253.852,A -85,B 0,C 180,E1 18016.75,E2 18016.75} C_VEL
LIN {X 0,Y 388.842,Z 250.863,A -85,B 0,C 180,E1 18015.665,E2 18015.665} C_VEL
LIN {X 0,Y 385.83,Z 248.32,A -85,B 0,C 180,E1 18013.793,E2 18013.793} C_VEL
LIN {X 0,Y 384.268,Z 244.981,A -85,B 0,C 180,E1 18012.396,E2 18012.396} C_VEL
LIN {X 0,Y 383.812,Z 244.424,A -85,B 0,C 180,E1 18012.029,E2 18012.029} C_VEL
LIN {X 0,Y 380.385,Z 241.855,A -85,B 0,C 180,E1 18009.227,E2 18009.227} C_VEL
LIN {X 0,Y 378.93,Z 238.588,A -85,B 0,C 180,E1 18007.353,E2 18007.353} C_VEL
LIN {X 0,Y 378.849,Z 237.983,A -85,B 0,C 180,E1 18006.973,E2 18006.973} C_VEL
LIN {X 0,Y 378.843,Z 238.041,A -85,B 0,C 180,E1 18002.874,E2 18002.874} C_VEL
LIN {X 0,Y 378.842,Z 237.977,A -85,B 0,C 180,E1 17998.79,E2 17998.79} C_VEL
LIN {X 0,Y 378.842,Z 237.999,A -85,B 0,C 180,E1 17994.7,E2 17994.7} C_VEL
LIN {X 0,Y 378.842,Z 238.004,A -85,B 0,C 180,E1 17990.735,E2 17990.735} C_VEL
LIN {X 0,Y 378.872,Z 238.232,A -85,B 0,C 180,E1 17988.661,E2 17988.661} C_VEL
LIN {X 0,Y 380.071,Z 241.43,A -85,B 0,C 180,E1 17987.85,E2 17987.85} C_VEL
LIN {X 0,Y 381.612,Z 243.662,A -85,B 0,C 180,E1 17987.131,E2 17987.131} C_VEL
LIN {X 0,Y 383.464,Z 247.268,A -85,B 0,C 180,E1 17986.12,E2 17986.12} C_VEL
LIN {X 0,Y 387.079,Z 254.192,A -85,B 0,C 180,E1 17984.262,E2 17984.262} C_VEL
LIN {X 0,Y 389.937,Z 259.625,A -85,B 0,C 180,E1 17982.849,E2 17982.849} C_VEL
LIN {X 0,Y 394.087,Z 267.357,A -85,B 0,C 180,E1 17980.895,E2 17980.895} C_VEL
LIN {X 0,Y 401.388,Z 281.511,A -85,B 0,C 180,E1 17977.596,E2 17977.596} C_VEL
LIN {X 0,Y 409.092,Z 296.602,A -85,B 0,C 180,E1 17974.366,E2 17974.366} C_VEL
LIN {X 0,Y 418.828,Z 316.5,A -85,B 0,C 180,E1 17970.541,E2 17970.541} C_VEL
LIN {X 0,Y 425.734,Z 330.733,A -85,B 0,C 180,E1 17968.1,E2 17968.1} C_VEL
LIN {X 0,Y 445.624,Z 361.563,A -85,B 0,C 180,E1 17964.863,E2 17964.863} C_VEL
LIN {X 0,Y 449.153,Z 367.707,A -85,B 0,C 180,E1 17964.297,E2 17964.297} C_VEL
LIN {X 0,Y 431.295,Z 623.048,A -85,B 0,C 180,E1 17959.116,E2 17959.116} C_VEL
LIN {X 0,Y 426.757,Z 693.714,A -85,B 0,C 180,E1 17957.627,E2 17957.627} C_VEL
LIN {X 0,Y 424.171,Z 718.167,A -85,B 0,C 180,E1 17956.898,E2 17956.898} C_VEL
LIN {X 0,Y 420.933,Z 742.907,A -85,B 0,C 180,E1 17955.926,E2 17955.926} C_VEL
LIN {X 0,Y 417.501,Z 765.209,A -85,B 0,C 180,E1 17954.825,E2 17954.825} C_VEL
LIN {X 0,Y 413.448,Z 788.171,A -85,B 0,C 180,E1 17953.429,E2 17953.429} C_VEL
LIN {X 0,Y 409.206,Z 810.052,A -85,B 0,C 180,E1 17951.841,E2 17951.841} C_VEL
LIN {X 0,Y 404.799,Z 830.866,A -85,B 0,C 180,E1 17950.028,E2 17950.028} C_VEL
LIN {X 0,Y 399.952,Z 852.42,A -85,B 0,C 180,E1 17947.813,E2 17947.813} C_VEL
LIN {X 0,Y 395.562,Z 871.48,A -85,B 0,C 180,E1 17945.517,E2 17945.517} C_VEL
LIN {X 0,Y 391.342,Z 889.34,A -85,B 0,C 180,E1 17942.971,E2 17942.971} C_VEL
LIN {X 0,Y 387.295,Z 906.832,A -85,B 0,C 180,E1 17940.056,E2 17940.056} C_VEL
LIN {X 0,Y 384.312,Z 920.375,A -85,B 0,C 180,E1 17937.42,E2 17937.42} C_VEL
LIN {X 0,Y 381.524,Z 934.074,A -85,B 0,C 180,E1 17934.297,E2 17934.297} C_VEL
LIN {X 0,Y 379.464,Z 945.788,A -85,B 0,C 180,E1 17931.161,E2 17931.161} C_VEL
LIN {X 0,Y 378.08,Z 955.501,A -85,B 0,C 180,E1 17928.024,E2 17928.024} C_VEL
LIN {X 0,Y 377.253,Z 963.595,A -85,B 0,C 180,E1 17924.898,E2 17924.898} C_VEL
LIN {X 0,Y 376.854,Z 970.579,A -85,B 0,C 180,E1 17921.478,E2 17921.478} C_VEL
LIN {X 0,Y 376.824,Z 974.966,A -85,B 0,C 180,E1 17918.699,E2 17918.699} C_VEL
LIN {X 0,Y 376.955,Z 978.678,A -85,B 0,C 180,E1 17915.48,E2 17915.48} C_VEL
LIN {X 0,Y 377.088,Z 980.675,A -85,B 0,C 180,E1 17912.279,E2 17912.279} C_VEL
LIN {X 0,Y 377.105,Z 981.226,A -85,B 0,C 180,E1 17909.544,E2 17909.544} C_VEL
LIN {X 0,Y 377.003,Z 980.629,A -85,B 0,C 180,E1 17906.655,E2 17906.655} C_VEL
LIN {X 0,Y 376.787,Z 978.379,A -85,B 0,C 180,E1 17903.295,E2 17903.295} C_VEL
LIN {X 0,Y 376.681,Z 974.912,A -85,B 0,C 180,E1 17900.219,E2 17900.219} C_VEL
LIN {X 0,Y 376.839,Z 969.657,A -85,B 0,C 180,E1 17896.809,E2 17896.809} C_VEL
LIN {X 0,Y 377.529,Z 962.292,A -85,B 0,C 180,E1 17893.22,E2 17893.22} C_VEL
LIN {X 0,Y 378.89,Z 953.664,A -85,B 0,C 180,E1 17889.775,E2 17889.775} C_VEL
LIN {X 0,Y 381.225,Z 942.664,A -85,B 0,C 180,E1 17886.177,E2 17886.177} C_VEL
LIN {X 0,Y 384.464,Z 930.371,A -85,B 0,C 180,E1 17882.759,E2 17882.759} C_VEL
LIN {X 0,Y 388.547,Z 916.635,A -85,B 0,C 180,E1 17879.538,E2 17879.538} C_VEL
LIN {X 0,Y 393.954,Z 900.197,A -85,B 0,C 180,E1 17876.231,E2 17876.231} C_VEL
LIN {X 0,Y 399.68,Z 883.887,A -85,B 0,C 180,E1 17873.423,E2 17873.423} C_VEL
LIN {X 0,Y 406.563,Z 864.805,A -85,B 0,C 180,E1 17870.616,E2 17870.616} C_VEL
LIN {X 0,Y 414.428,Z 843.55,A -85,B 0,C 180,E1 17867.97,E2 17867.97} C_VEL
LIN {X 0,Y 422.162,Z 822.68,A -85,B 0,C 180,E1 17865.771,E2 17865.771} C_VEL
LIN {X 0,Y 430.479,Z 799.67,A -85,B 0,C 180,E1 17863.749,E2 17863.749} C_VEL
LIN {X 0,Y 439.113,Z 775.1,A -85,B 0,C 180,E1 17861.973,E2 17861.973} C_VEL
LIN {X 0,Y 447.335,Z 750.521,A -85,B 0,C 180,E1 17860.538,E2 17860.538} C_VEL
LIN {X 0,Y 454.928,Z 726.213,A -85,B 0,C 180,E1 17859.415,E2 17859.415} C_VEL
LIN {X 0,Y 462.044,Z 701.016,A -85,B 0,C 180,E1 17858.528,E2 17858.528} C_VEL
LIN {X 0,Y 467.431,Z 678.924,A -85,B 0,C 180,E1 17857.908,E2 17857.908} C_VEL
LIN {X 0,Y 460.127,Z 703.41,A -85,B 0,C 180,E1 17857.087,E2 17857.087} C_VEL
LIN {X 0,Y 452.805,Z 723.987,A -85,B 0,C 180,E1 17856.207,E2 17856.207} C_VEL
LIN {X 0,Y 444.322,Z 745.531,A -85,B 0,C 180,E1 17855.019,E2 17855.019} C_VEL
LIN {X 0,Y 435.095,Z 767.549,A -85,B 0,C 180,E1 17853.473,E2 17853.473} C_VEL
LIN {X 0,Y 425.825,Z 789.229,A -85,B 0,C 180,E1 17851.576,E2 17851.576} C_VEL
LIN {X 0,Y 417.313,Z 809.369,A -85,B 0,C 180,E1 17849.419,E2 17849.419} C_VEL
LIN {X 0,Y 409.631,Z 828.003,A -85,B 0,C 180,E1 17847.002,E2 17847.002} C_VEL
LIN {X 0,Y 403.38,Z 843.309,A -85,B 0,C 180,E1 17844.61,E2 17844.61} C_VEL
LIN {X 0,Y 397.742,Z 857.099,A -85,B 0,C 180,E1 17841.998,E2 17841.998} C_VEL
LIN {X 0,Y 393.218,Z 868.031,A -85,B 0,C 180,E1 17839.458,E2 17839.458} C_VEL
LIN {X 0,Y 389.213,Z 877.396,A -85,B 0,C 180,E1 17836.722,E2 17836.722} C_VEL
LIN {X 0,Y 386.092,Z 884.31,A -85,B 0,C 180,E1 17834.09,E2 17834.09} C_VEL
LIN {X 0,Y 383.585,Z 889.38,A -85,B 0,C 180,E1 17831.426,E2 17831.426} C_VEL
LIN {X 0,Y 381.549,Z 892.794,A -85,B 0,C 180,E1 17828.591,E2 17828.591} C_VEL
LIN {X 0,Y 380.19,Z 894.18,A -85,B 0,C 180,E1 17826.039,E2 17826.039} C_VEL
LIN {X 0,Y 379.178,Z 894.027,A -85,B 0,C 180,E1 17823.326,E2 17823.326} C_VEL
LIN {X 0,Y 378.542,Z 892.117,A -85,B 0,C 180,E1 17820.605,E2 17820.605} C_VEL
LIN {X 0,Y 378.201,Z 888.493,A -85,B 0,C 180,E1 17817.879,E2 17817.879} C_VEL
LIN {X 0,Y 378.151,Z 883.073,A -85,B 0,C 180,E1 17815.146,E2 17815.146} C_VEL
LIN {X 0,Y 378.383,Z 876.257,A -85,B 0,C 180,E1 17812.56,E2 17812.56} C_VEL
LIN {X 0,Y 378.947,Z 866.932,A -85,B 0,C 180,E1 17809.802,E2 17809.802} C_VEL
LIN {X 0,Y 379.849,Z 856.175,A -85,B 0,C 180,E1 17807.225,E2 17807.225} C_VEL
LIN {X 0,Y 381.079,Z 843.917,A -85,B 0,C 180,E1 17804.788,E2 17804.788} C_VEL
LIN {X 0,Y 382.655,Z 829.783,A -85,B 0,C 180,E1 17802.434,E2 17802.434} C_VEL
LIN {X 0,Y 384.504,Z 814.134,A -85,B 0,C 180,E1 17800.241,E2 17800.241} C_VEL
LIN {X 0,Y 386.67,Z 796.201,A -85,B 0,C 180,E1 17798.138,E2 17798.138} C_VEL
LIN {X 0,Y 388.93,Z 777.179,A -85,B 0,C 180,E1 17796.275,E2 17796.275} C_VEL
LIN {X 0,Y 391.231,Z 757.207,A -85,B 0,C 180,E1 17794.654,E2 17794.654} C_VEL
LIN {X 0,Y 393.485,Z 736.399,A -85,B 0,C 180,E1 17793.27,E2 17793.27} C_VEL
LIN {X 0,Y 395.641,Z 713.888,A -85,B 0,C 180,E1 17792.084,E2 17792.084} C_VEL
LIN {X 0,Y 397.561,Z 690.842,A -85,B 0,C 180,E1 17791.161,E2 17791.161} C_VEL
LIN {X 0,Y 399.673,Z 658.334,A -85,B 0,C 180,E1 17790.236,E2 17790.236} C_VEL
LIN {X 0,Y 409.338,Z 509.956,A -85,B 0,C 180,E1 17786.421,E2 17786.421} C_VEL
LIN {X 0,Y 404.878,Z 434.229,A -85,B 0,C 180,E1 17783.651,E2 17783.651} C_VEL
LIN {X 0,Y 408.253,Z 410.899,A -85,B 0,C 180,E1 17781.586,E2 17781.586} C_VEL
LIN {X 0,Y 410.174,Z 410.673,A -85,B 0,C 180,E1 17781.208,E2 17781.208} C_VEL
LIN {X 0,Y 413.693,Z 408.067,A -85,B 0,C 180,E1 17780.709,E2 17780.709} C_VEL
LIN {X 0,Y 417.643,Z 403.908,A -85,B 0,C 180,E1 17780.265,E2 17780.265} C_VEL
LIN {X 0,Y 420.991,Z 402.172,A -85,B 0,C 180,E1 17779.757,E2 17779.757} C_VEL
LIN {X 0,Y 425.545,Z 398.227,A -85,B 0,C 180,E1 17779.216,E2 17779.216} C_VEL
LIN {X 0,Y 427.093,Z 396.825,A -85,B 0,C 180,E1 17779.04,E2 17779.04} C_VEL
LIN {X 0,Y 432.087,Z 393.697,A -85,B 0,C 180,E1 17778.383,E2 17778.383} C_VEL
LIN {X 0,Y 436.002,Z 390.332,A -85,B 0,C 180,E1 17777.96,E2 17777.96} C_VEL
LIN {X 0,Y 441.889,Z 386.617,A -85,B 0,C 180,E1 17777.247,E2 17777.247} C_VEL
LIN {X 0,Y 445.028,Z 384.06,A -85,B 0,C 180,E1 17776.919,E2 17776.919} C_VEL
LIN {X 0,Y 447.297,Z 382.973,A -85,B 0,C 180,E1 17776.632,E2 17776.632} C_VEL
LIN {X 0,Y 441.667,Z 409.03,A -85,B 0,C 180,E1 17775.71,E2 17775.71} C_VEL
LIN {X 0,Y 437.314,Z 489.547,A -85,B 0,C 180,E1 17774.329,E2 17774.329} C_VEL
LIN {X 0,Y 432.777,Z 549.361,A -85,B 0,C 180,E1 17773.085,E2 17773.085} C_VEL
LIN {X 0,Y 426.969,Z 611.022,A -85,B 0,C 180,E1 17771.577,E2 17771.577} C_VEL
LIN {X 0,Y 422.69,Z 655.453,A -85,B 0,C 180,E1 17770.281,E2 17770.281} C_VEL
LIN {X 0,Y 420.372,Z 682.454,A -85,B 0,C 180,E1 17769.311,E2 17769.311} C_VEL
LIN {X 0,Y 418.051,Z 702.567,A -85,B 0,C 180,E1 17768.362,E2 17768.362} C_VEL
LIN {X 0,Y 414.965,Z 723.485,A -85,B 0,C 180,E1 17767.12,E2 17767.12} C_VEL
LIN {X 0,Y 411.486,Z 743.206,A -85,B 0,C 180,E1 17765.675,E2 17765.675} C_VEL
LIN {X 0,Y 407.506,Z 762.686,A -85,B 0,C 180,E1 17763.941,E2 17763.941} C_VEL
LIN {X 0,Y 403.42,Z 780.555,A -85,B 0,C 180,E1 17762.033,E2 17762.033} C_VEL
LIN {X 0,Y 399.115,Z 797.862,A -85,B 0,C 180,E1 17759.821,E2 17759.821} C_VEL
LIN {X 0,Y 394.99,Z 813.492,A -85,B 0,C 180,E1 17757.434,E2 17757.434} C_VEL
LIN {X 0,Y 391.041,Z 827.948,A -85,B 0,C 180,E1 17754.794,E2 17754.794} C_VEL
LIN {X 0,Y 387.496,Z 840.784,A -85,B 0,C 180,E1 17751.972,E2 17751.972} C_VEL
LIN {X 0,Y 384.448,Z 852.02,A -85,B 0,C 180,E1 17748.972,E2 17748.972} C_VEL
LIN {X 0,Y 382.074,Z 861.207,A -85,B 0,C 180,E1 17745.949,E2 17745.949} C_VEL
LIN {X 0,Y 380.731,Z 866.883,A -85,B 0,C 180,E1 17743.688,E2 17743.688} C_VEL
LIN {X 0,Y 379.21,Z 869.447,A -85,B 0,C 180,E1 17742.604,E2 17742.604} C_VEL
LIN {X 0,Y 371.898,Z 875.806,A -85,B 0,C 180,E1 17739.717,E2 17739.717} C_VEL
LIN {X 0,Y 370.852,Z 877.297,A -85,B 0,C 180,E1 17738.727,E2 17738.727} C_VEL
LIN {X 0,Y 370.201,Z 880.928,A -85,B 0,C 180,E1 17735.425,E2 17735.425} C_VEL
LIN {X 0,Y 369.888,Z 882.807,A -85,B 0,C 180,E1 17732.169,E2 17732.169} C_VEL
LIN {X 0,Y 369.83,Z 883.108,A -85,B 0,C 180,E1 17729.071,E2 17729.071} C_VEL
LIN {X 0,Y 370.03,Z 881.872,A -85,B 0,C 180,E1 17725.816,E2 17725.816} C_VEL
LIN {X 0,Y 370.54,Z 879.03,A -85,B 0,C 180,E1 17722.558,E2 17722.558} C_VEL
LIN {X 0,Y 371.46,Z 874.454,A -85,B 0,C 180,E1 17719.267,E2 17719.267} C_VEL
LIN {X 0,Y 372.927,Z 868.165,A -85,B 0,C 180,E1 17716.036,E2 17716.036} C_VEL
LIN {X 0,Y 374.905,Z 860.388,A -85,B 0,C 180,E1 17712.94,E2 17712.94} C_VEL
LIN {X 0,Y 377.56,Z 850.76,A -85,B 0,C 180,E1 17709.862,E2 17709.862} C_VEL
LIN {X 0,Y 380.727,Z 839.683,A -85,B 0,C 180,E1 17706.964,E2 17706.964} C_VEL
LIN {X 0,Y 384.34,Z 827.194,A -85,B 0,C 180,E1 17704.249,E2 17704.249} C_VEL
LIN {X 0,Y 388.302,Z 813.313,A -85,B 0,C 180,E1 17701.718,E2 17701.718} C_VEL
LIN {X 0,Y 392.51,Z 798.005,A -85,B 0,C 180,E1 17699.371,E2 17699.371} C_VEL
LIN {X 0,Y 396.862,Z 781.154,A -85,B 0,C 180,E1 17697.201,E2 17697.201} C_VEL
LIN {X 0,Y 401.131,Z 763.186,A -85,B 0,C 180,E1 17695.265,E2 17695.265} C_VEL
LIN {X 0,Y 405.254,Z 743.612,A -85,B 0,C 180,E1 17693.514,E2 17693.514} C_VEL
LIN {X 0,Y 408.889,Z 723.656,A -85,B 0,C 180,E1 17692.047,E2 17692.047} C_VEL
LIN {X 0,Y 412.071,Z 702.557,A -85,B 0,C 180,E1 17690.795,E2 17690.795} C_VEL
LIN {X 0,Y 414.643,Z 680.459,A -85,B 0,C 180,E1 17689.768,E2 17689.768} C_VEL
LIN {X 0,Y 417.74,Z 645.31,A -85,B 0,C 180,E1 17688.561,E2 17688.561} C_VEL
LIN {X 0,Y 423.364,Z 590.497,A -85,B 0,C 180,E1 17687.039,E2 17687.039} C_VEL
LIN {X 0,Y 428.981,Z 528.55,A -85,B 0,C 180,E1 17685.598,E2 17685.598} C_VEL
LIN {X 0,Y 432.839,Z 473.766,A -85,B 0,C 180,E1 17684.519,E2 17684.519} C_VEL
LIN {X 0,Y 436.393,Z 409.894,A -85,B 0,C 180,E1 17683.421,E2 17683.421} C_VEL
LIN {X 0,Y 443.125,Z 379.736,A -85,B 0,C 180,E1 17682.307,E2 17682.307} C_VEL
LIN {X 0,Y 443.418,Z 370.191,A -85,B 0,C 180,E1 17681.613,E2 17681.613} C_VEL
LIN {X 0,Y 436.975,Z 351.876,A -85,B 0,C 180,E1 17678.996,E2 17678.996} C_VEL
LIN {X 0,Y 430.35,Z 335.39,A -85,B 0,C 180,E1 17676.333,E2 17676.333} C_VEL
LIN {X 0,Y 423.53,Z 320.133,A -85,B 0,C 180,E1 17673.535,E2 17673.535} C_VEL
LIN {X 0,Y 416.8,Z 306.982,A -85,B 0,C 180,E1 17670.814,E2 17670.814} C_VEL
LIN {X 0,Y 410.43,Z 295.258,A -85,B 0,C 180,E1 17668.047,E2 17668.047} C_VEL
LIN {X 0,Y 404.335,Z 285.234,A -85,B 0,C 180,E1 17665.329,E2 17665.329} C_VEL
LIN {X 0,Y 400.776,Z 279.844,A -85,B 0,C 180,E1 17663.706,E2 17663.706} C_VEL
LIN {X 0,Y 397.678,Z 275.026,A -85,B 0,C 180,E1 17662.157,E2 17662.157} C_VEL
LIN {X 0,Y 394.835,Z 270.674,A -85,B 0,C 180,E1 17660.649,E2 17660.649} C_VEL
LIN {X 0,Y 391.2,Z 265.823,A -85,B 0,C 180,E1 17658.671,E2 17658.671} C_VEL
LIN {X 0,Y 390.26,Z 264.119,A -85,B 0,C 180,E1 17658.06,E2 17658.06} C_VEL
LIN {X 0,Y 387.368,Z 260.8,A -85,B 0,C 180,E1 17656.341,E2 17656.341} C_VEL
LIN {X 0,Y 386.217,Z 258.366,A -85,B 0,C 180,E1 17655.466,E2 17655.466} C_VEL
LIN {X 0,Y 383.219,Z 255.642,A -85,B 0,C 180,E1 17653.505,E2 17653.505} C_VEL
LIN {X 0,Y 381.584,Z 252.095,A -85,B 0,C 180,E1 17651.947,E2 17651.947} C_VEL
LIN {X 0,Y 378.174,Z 249.532,A -85,B 0,C 180,E1 17649.128,E2 17649.128} C_VEL
LIN {X 0,Y 376.726,Z 246.121,A -85,B 0,C 180,E1 17647.089,E2 17647.089} C_VEL
LIN {X 0,Y 376.458,Z 245.616,A -85,B 0,C 180,E1 17646.711,E2 17646.711} C_VEL
LIN {X 0,Y 372.699,Z 243.102,A -85,B 0,C 180,E1 17638.77,E2 17638.77} C_VEL
LIN {X 0,Y 373.273,Z 243.735,A -85,B 0,C 180,E1 17634.158,E2 17634.158} C_VEL
LIN {X 0,Y 376.455,Z 245.92,A -85,B 0,C 180,E1 17628.975,E2 17628.975} C_VEL
LIN {X 0,Y 376.938,Z 248.999,A -85,B 0,C 180,E1 17627.903,E2 17627.903} C_VEL
LIN {X 0,Y 377.372,Z 250.956,A -85,B 0,C 180,E1 17627.176,E2 17627.176} C_VEL
LIN {X 0,Y 378.09,Z 252.989,A -85,B 0,C 180,E1 17626.387,E2 17626.387} C_VEL
LIN {X 0,Y 381.942,Z 260.443,A -85,B 0,C 180,E1 17624.357,E2 17624.357} C_VEL
LIN {X 0,Y 386.64,Z 269.178,A -85,B 0,C 180,E1 17622.076,E2 17622.076} C_VEL
LIN {X 0,Y 393.585,Z 282.568,A -85,B 0,C 180,E1 17618.854,E2 17618.854} C_VEL
LIN {X 0,Y 401.935,Z 299.062,A -85,B 0,C 180,E1 17615.231,E2 17615.231} C_VEL
LIN {X 0,Y 410.782,Z 317.019,A -85,B 0,C 180,E1 17611.663,E2 17611.663} C_VEL
LIN {X 0,Y 417.869,Z 331.617,A -85,B 0,C 180,E1 17609.059,E2 17609.059} C_VEL
LIN {X 0,Y 436.305,Z 360.278,A -85,B 0,C 180,E1 17605.941,E2 17605.941} C_VEL
LIN {X 0,Y 442.82,Z 370.929,A -85,B 0,C 180,E1 17604.902,E2 17604.902} C_VEL
LIN {X 0,Y 425.049,Z 615.432,A -85,B 0,C 180,E1 17599.852,E2 17599.852} C_VEL
LIN {X 0,Y 419.838,Z 693.71,A -85,B 0,C 180,E1 17598.171,E2 17598.171} C_VEL
LIN {X 0,Y 417.204,Z 717.985,A -85,B 0,C 180,E1 17597.434,E2 17597.434} C_VEL
LIN {X 0,Y 413.793,Z 743.335,A -85,B 0,C 180,E1 17596.419,E2 17596.419} C_VEL
LIN {X 0,Y 410.214,Z 765.969,A -85,B 0,C 180,E1 17595.278,E2 17595.278} C_VEL
LIN {X 0,Y 406.115,Z 788.494,A -85,B 0,C 180,E1 17593.874,E2 17593.874} C_VEL
LIN {X 0,Y 401.696,Z 810.64,A -85,B 0,C 180,E1 17592.227,E2 17592.227} C_VEL
LIN {X 0,Y 397.243,Z 831.201,A -85,B 0,C 180,E1 17590.402,E2 17590.402} C_VEL
LIN {X 0,Y 392.5,Z 851.807,A -85,B 0,C 180,E1 17588.246,E2 17588.246} C_VEL
LIN {X 0,Y 388.001,Z 870.876,A -85,B 0,C 180,E1 17585.915,E2 17585.915} C_VEL
LIN {X 0,Y 383.726,Z 888.522,A -85,B 0,C 180,E1 17583.354,E2 17583.354} C_VEL
LIN {X 0,Y 379.566,Z 906.051,A -85,B 0,C 180,E1 17580.383,E2 17580.383} C_VEL
LIN {X 0,Y 376.502,Z 919.634,A -85,B 0,C 180,E1 17577.694,E2 17577.694} C_VEL
LIN {X 0,Y 373.64,Z 933.36,A -85,B 0,C 180,E1 17574.506,E2 17574.506} C_VEL
LIN {X 0,Y 371.584,Z 944.731,A -85,B 0,C 180,E1 17571.401,E2 17571.401} C_VEL
LIN {X 0,Y 370.123,Z 954.76,A -85,B 0,C 180,E1 17568.1,E2 17568.1} C_VEL
LIN {X 0,Y 369.274,Z 963.009,A -85,B 0,C 180,E1 17564.837,E2 17564.837} C_VEL
LIN {X 0,Y 368.9,Z 969.788,A -85,B 0,C 180,E1 17561.412,E2 17561.412} C_VEL
LIN {X 0,Y 368.885,Z 974.143,A -85,B 0,C 180,E1 17558.574,E2 17558.574} C_VEL
LIN {X 0,Y 369.026,Z 977.784,A -85,B 0,C 180,E1 17555.286,E2 17555.286} C_VEL
LIN {X 0,Y 369.163,Z 979.66,A -85,B 0,C 180,E1 17552.173,E2 17552.173} C_VEL
LIN {X 0,Y 369.166,Z 980.199,A -85,B 0,C 180,E1 17549.379,E2 17549.379} C_VEL
LIN {X 0,Y 369.057,Z 979.635,A -85,B 0,C 180,E1 17546.583,E2 17546.583} C_VEL
LIN {X 0,Y 368.807,Z 977.464,A -85,B 0,C 180,E1 17543.149,E2 17543.149} C_VEL
LIN {X 0,Y 368.697,Z 973.817,A -85,B 0,C 180,E1 17539.847,E2 17539.847} C_VEL
LIN {X 0,Y 368.887,Z 968.537,A -85,B 0,C 180,E1 17536.36,E2 17536.36} C_VEL
LIN {X 0,Y 369.681,Z 961.169,A -85,B 0,C 180,E1 17532.691,E2 17532.691} C_VEL
LIN {X 0,Y 371.108,Z 952.958,A -85,B 0,C 180,E1 17529.331,E2 17529.331} C_VEL
LIN {X 0,Y 373.613,Z 942.104,A -85,B 0,C 180,E1 17525.66,E2 17525.66} C_VEL
LIN {X 0,Y 377.059,Z 929.949,A -85,B 0,C 180,E1 17522.178,E2 17522.178} C_VEL
LIN {X 0,Y 381.621,Z 915.732,A -85,B 0,C 180,E1 17518.749,E2 17518.749} C_VEL
LIN {X 0,Y 387.402,Z 899.481,A -85,B 0,C 180,E1 17515.401,E2 17515.401} C_VEL
LIN {X 0,Y 393.749,Z 882.654,A -85,B 0,C 180,E1 17512.45,E2 17512.45} C_VEL
LIN {X 0,Y 401.166,Z 863.625,A -85,B 0,C 180,E1 17509.606,E2 17509.606} C_VEL
LIN {X 0,Y 409.288,Z 843.31,A -85,B 0,C 180,E1 17507.031,E2 17507.031} C_VEL
LIN {X 0,Y 417.921,Z 821.672,A -85,B 0,C 180,E1 17504.717,E2 17504.717} C_VEL
LIN {X 0,Y 427.008,Z 798.545,A -85,B 0,C 180,E1 17502.67,E2 17502.67} C_VEL
LIN {X 0,Y 436.125,Z 774.699,A -85,B 0,C 180,E1 17500.936,E2 17500.936} C_VEL
LIN {X 0,Y 445.112,Z 750.099,A -85,B 0,C 180,E1 17499.499,E2 17499.499} C_VEL
LIN {X 0,Y 453.088,Z 726.812,A -85,B 0,C 180,E1 17498.424,E2 17498.424} C_VEL
LIN {X 0,Y 458.046,Z 711.057,A -85,B 0,C 180,E1 17497.837,E2 17497.837} C_VEL
LIN {X 0,Y 449.744,Z 732.033,A -85,B 0,C 180,E1 17496.89,E2 17496.89} C_VEL
LIN {X 0,Y 440.64,Z 752.821,A -85,B 0,C 180,E1 17495.675,E2 17495.675} C_VEL
LIN {X 0,Y 431.017,Z 773.396,A -85,B 0,C 180,E1 17494.153,E2 17494.153} C_VEL
LIN {X 0,Y 421.296,Z 793.853,A -85,B 0,C 180,E1 17492.277,E2 17492.277} C_VEL
LIN {X 0,Y 412.313,Z 813.002,A -85,B 0,C 180,E1 17490.132,E2 17490.132} C_VEL
LIN {X 0,Y 404.141,Z 830.82,A -85,B 0,C 180,E1 17487.719,E2 17487.719} C_VEL
LIN {X 0,Y 397.131,Z 846.339,A -85,B 0,C 180,E1 17485.183,E2 17485.183} C_VEL
LIN {X 0,Y 391.155,Z 859.621,A -85,B 0,C 180,E1 17482.547,E2 17482.547} C_VEL
LIN {X 0,Y 386.349,Z 870.2,A -85,B 0,C 180,E1 17479.976,E2 17479.976} C_VEL
LIN {X 0,Y 382.158,Z 879.13,A -85,B 0,C 180,E1 17477.254,E2 17477.254} C_VEL
LIN {X 0,Y 378.757,Z 886.02,A -85,B 0,C 180,E1 17474.524,E2 17474.524} C_VEL
LIN {X 0,Y 375.938,Z 891.148,A -85,B 0,C 180,E1 17471.662,E2 17471.662} C_VEL
LIN {X 0,Y 373.877,Z 894.196,A -85,B 0,C 180,E1 17468.923,E2 17468.923} C_VEL
LIN {X 0,Y 372.344,Z 895.519,A -85,B 0,C 180,E1 17466.166,E2 17466.166} C_VEL
LIN {X 0,Y 371.268,Z 895.139,A -85,B 0,C 180,E1 17463.397,E2 17463.397} C_VEL
LIN {X 0,Y 370.597,Z 893.05,A -85,B 0,C 180,E1 17460.618,E2 17460.618} C_VEL
LIN {X 0,Y 370.227,Z 888.959,A -85,B 0,C 180,E1 17457.678,E2 17457.678} C_VEL
LIN {X 0,Y 370.195,Z 883.259,A -85,B 0,C 180,E1 17454.886,E2 17454.886} C_VEL
LIN {X 0,Y 370.477,Z 875.638,A -85,B 0,C 180,E1 17452.088,E2 17452.088} C_VEL
LIN {X 0,Y 371.115,Z 865.96,A -85,B 0,C 180,E1 17449.286,E2 17449.286} C_VEL
LIN {X 0,Y 372.157,Z 854.294,A -85,B 0,C 180,E1 17446.557,E2 17446.557} C_VEL
LIN {X 0,Y 373.557,Z 841.04,A -85,B 0,C 180,E1 17443.996,E2 17443.996} C_VEL
LIN {X 0,Y 375.292,Z 826.18,A -85,B 0,C 180,E1 17441.596,E2 17441.596} C_VEL
LIN {X 0,Y 377.313,Z 809.736,A -85,B 0,C 180,E1 17439.362,E2 17439.362} C_VEL
LIN {X 0,Y 379.573,Z 791.584,A -85,B 0,C 180,E1 17437.299,E2 17437.299} C_VEL
LIN {X 0,Y 381.887,Z 772.406,A -85,B 0,C 180,E1 17435.481,E2 17435.481} C_VEL
LIN {X 0,Y 384.23,Z 752.327,A -85,B 0,C 180,E1 17433.909,E2 17433.909} C_VEL
LIN {X 0,Y 386.651,Z 729.773,A -85,B 0,C 180,E1 17432.478,E2 17432.478} C_VEL
LIN {X 0,Y 388.821,Z 706.949,A -85,B 0,C 180,E1 17431.34,E2 17431.34} C_VEL
LIN {X 0,Y 390.726,Z 683.562,A -85,B 0,C 180,E1 17430.473,E2 17430.473} C_VEL
LIN {X 0,Y 402.308,Z 510.821,A -85,B 0,C 180,E1 17425.891,E2 17425.891} C_VEL
LIN {X 0,Y 398.01,Z 433.158,A -85,B 0,C 180,E1 17422.982,E2 17422.982} C_VEL
LIN {X 0,Y 399.122,Z 425.775,A -85,B 0,C 180,E1 17422.318,E2 17422.318} C_VEL
LIN {X 0,Y 400.794,Z 425.672,A -85,B 0,C 180,E1 17421.96,E2 17421.96} C_VEL
LIN {X 0,Y 404.192,Z 423.194,A -85,B 0,C 180,E1 17421.435,E2 17421.435} C_VEL
LIN {X 0,Y 408.518,Z 418.349,A -85,B 0,C 180,E1 17420.931,E2 17420.931} C_VEL
LIN {X 0,Y 412.157,Z 416.376,A -85,B 0,C 180,E1 17420.354,E2 17420.354} C_VEL
LIN {X 0,Y 416.658,Z 412.281,A -85,B 0,C 180,E1 17419.793,E2 17419.793} C_VEL
LIN {X 0,Y 418.233,Z 410.69,A -85,B 0,C 180,E1 17419.617,E2 17419.617} C_VEL
LIN {X 0,Y 423.151,Z 407.544,A -85,B 0,C 180,E1 17418.936,E2 17418.936} C_VEL
LIN {X 0,Y 427.767,Z 403.435,A -85,B 0,C 180,E1 17418.406,E2 17418.406} C_VEL
LIN {X 0,Y 433.627,Z 399.518,A -85,B 0,C 180,E1 17417.676,E2 17417.676} C_VEL
LIN {X 0,Y 436.753,Z 396.908,A -85,B 0,C 180,E1 17417.339,E2 17417.339} C_VEL
LIN {X 0,Y 439.482,Z 395.295,A -85,B 0,C 180,E1 17417,E2 17417} C_VEL
LIN {X 0,Y 436.048,Z 411.878,A -85,B 0,C 180,E1 17416.427,E2 17416.427} C_VEL
LIN {X 0,Y 431.592,Z 491.845,A -85,B 0,C 180,E1 17415.044,E2 17415.044} C_VEL
LIN {X 0,Y 426.935,Z 551.477,A -85,B 0,C 180,E1 17413.794,E2 17413.794} C_VEL
LIN {X 0,Y 421.004,Z 612.454,A -85,B 0,C 180,E1 17412.283,E2 17412.283} C_VEL
LIN {X 0,Y 416.613,Z 656.627,A -85,B 0,C 180,E1 17410.976,E2 17410.976} C_VEL
LIN {X 0,Y 414.143,Z 684.167,A -85,B 0,C 180,E1 17409.969,E2 17409.969} C_VEL
LIN {X 0,Y 411.671,Z 704.67,A -85,B 0,C 180,E1 17408.982,E2 17408.982} C_VEL
LIN {X 0,Y 408.494,Z 725.351,A -85,B 0,C 180,E1 17407.73,E2 17407.73} C_VEL
LIN {X 0,Y 404.886,Z 745.039,A -85,B 0,C 180,E1 17406.261,E2 17406.261} C_VEL
LIN {X 0,Y 400.919,Z 763.783,A -85,B 0,C 180,E1 17404.568,E2 17404.568} C_VEL
LIN {X 0,Y 396.544,Z 782.178,A -85,B 0,C 180,E1 17402.571,E2 17402.571} C_VEL
LIN {X 0,Y 392.084,Z 799.399,A -85,B 0,C 180,E1 17400.327,E2 17400.327} C_VEL
LIN {X 0,Y 387.682,Z 815.388,A -85,B 0,C 180,E1 17397.829,E2 17397.829} C_VEL
LIN {X 0,Y 383.596,Z 829.715,A -85,B 0,C 180,E1 17395.143,E2 17395.143} C_VEL
LIN {X 0,Y 379.924,Z 842.44,A -85,B 0,C 180,E1 17392.271,E2 17392.271} C_VEL
LIN {X 0,Y 376.762,Z 853.567,A -85,B 0,C 180,E1 17389.213,E2 17389.213} C_VEL
LIN {X 0,Y 374.193,Z 863.077,A -85,B 0,C 180,E1 17385.976,E2 17385.976} C_VEL
LIN {X 0,Y 372.324,Z 870.574,A -85,B 0,C 180,E1 17382.722,E2 17382.722} C_VEL
LIN {X 0,Y 371.08,Z 876.131,A -85,B 0,C 180,E1 17379.527,E2 17379.527} C_VEL
LIN {X 0,Y 370.852,Z 877.297,A -85,B 0,C 180,E1 17378.727,E2 17378.727} C_VEL
LIN {X 0,Y 369.576,Z 878.907,A -85,B 0,C 180,E1 17377.566,E2 17377.566} C_VEL
LIN {X 0,Y 362.889,Z 882.676,A -85,B 0,C 180,E1 17374.46,E2 17374.46} C_VEL
LIN {X 0,Y 362.034,Z 883.325,A -85,B 0,C 180,E1 17373.417,E2 17373.417} C_VEL
LIN {X 0,Y 361.899,Z 884.203,A -85,B 0,C 180,E1 17370.158,E2 17370.158} C_VEL
LIN {X 0,Y 361.99,Z 883.531,A -85,B 0,C 180,E1 17366.992,E2 17366.992} C_VEL
LIN {X 0,Y 362.391,Z 881.282,A -85,B 0,C 180,E1 17363.664,E2 17363.664} C_VEL
LIN {X 0,Y 363.134,Z 877.643,A -85,B 0,C 180,E1 17360.491,E2 17360.491} C_VEL
LIN {X 0,Y 364.434,Z 872.141,A -85,B 0,C 180,E1 17357.16,E2 17357.16} C_VEL
LIN {X 0,Y 366.359,Z 864.769,A -85,B 0,C 180,E1 17353.836,E2 17353.836} C_VEL
LIN {X 0,Y 369.008,Z 855.422,A -85,B 0,C 180,E1 17350.532,E2 17350.532} C_VEL
LIN {X 0,Y 372.088,Z 845.046,A -85,B 0,C 180,E1 17347.568,E2 17347.568} C_VEL
LIN {X 0,Y 375.623,Z 833.33,A -85,B 0,C 180,E1 17344.792,E2 17344.792} C_VEL
LIN {X 0,Y 379.769,Z 819.481,A -85,B 0,C 180,E1 17342.053,E2 17342.053} C_VEL
LIN {X 0,Y 384.109,Z 804.526,A -85,B 0,C 180,E1 17339.582,E2 17339.582} C_VEL
LIN {X 0,Y 388.694,Z 787.801,A -85,B 0,C 180,E1 17337.266,E2 17337.266} C_VEL
LIN {X 0,Y 393.15,Z 770.226,A -85,B 0,C 180,E1 17335.234,E2 17335.234} C_VEL
LIN {X 0,Y 397.486,Z 751.2,A -85,B 0,C 180,E1 17333.403,E2 17333.403} C_VEL
LIN {X 0,Y 401.362,Z 731.573,A -85,B 0,C 180,E1 17331.842,E2 17331.842} C_VEL
LIN {X 0,Y 404.643,Z 712.102,A -85,B 0,C 180,E1 17330.576,E2 17330.576} C_VEL
LIN {X 0,Y 407.411,Z 691.583,A -85,B 0,C 180,E1 17329.499,E2 17329.499} C_VEL
LIN {X 0,Y 409.614,Z 669.832,A -85,B 0,C 180,E1 17328.619,E2 17328.619} C_VEL
LIN {X 0,Y 413.811,Z 626.601,A -85,B 0,C 180,E1 17327.242,E2 17327.242} C_VEL
LIN {X 0,Y 419.839,Z 568.778,A -85,B 0,C 180,E1 17325.731,E2 17325.731} C_VEL
LIN {X 0,Y 424.984,Z 508.898,A -85,B 0,C 180,E1 17324.409,E2 17324.409} C_VEL
LIN {X 0,Y 428.551,Z 453.272,A -85,B 0,C 180,E1 17323.382,E2 17323.382} C_VEL
LIN {X 0,Y 430.849,Z 412.705,A -85,B 0,C 180,E1 17322.685,E2 17322.685} C_VEL
LIN {X 0,Y 437.854,Z 381.493,A -85,B 0,C 180,E1 17321.543,E2 17321.543} C_VEL
LIN {X 0,Y 438.102,Z 374.288,A -85,B 0,C 180,E1 17321.009,E2 17321.009} C_VEL
LIN {X 0,Y 431.7,Z 356.101,A -85,B 0,C 180,E1 17318.37,E2 17318.37} C_VEL
LIN {X 0,Y 425.544,Z 340.551,A -85,B 0,C 180,E1 17315.808,E2 17315.808} C_VEL
LIN {X 0,Y 418.875,Z 325.42,A -85,B 0,C 180,E1 17312.974,E2 17312.974} C_VEL
LIN {X 0,Y 411.539,Z 310.81,A -85,B 0,C 180,E1 17309.873,E2 17309.873} C_VEL
LIN {X 0,Y 405.656,Z 300.356,A -85,B 0,C 180,E1 17307.288,E2 17307.288} C_VEL
LIN {X 0,Y 401.04,Z 292.309,A -85,B 0,C 180,E1 17305.078,E2 17305.078} C_VEL
LIN {X 0,Y 397.213,Z 286.474,A -85,B 0,C 180,E1 17303.279,E2 17303.279} C_VEL
LIN {X 0,Y 394.441,Z 281.986,A -85,B 0,C 180,E1 17301.8,E2 17301.8} C_VEL
LIN {X 0,Y 391.017,Z 276.874,A -85,B 0,C 180,E1 17299.961,E2 17299.961} C_VEL
LIN {X 0,Y 388.14,Z 272.719,A -85,B 0,C 180,E1 17298.279,E2 17298.279} C_VEL
LIN {X 0,Y 387.304,Z 271.349,A -85,B 0,C 180,E1 17297.736,E2 17297.736} C_VEL
LIN {X 0,Y 384.465,Z 267.744,A -85,B 0,C 180,E1 17295.925,E2 17295.925} C_VEL
LIN {X 0,Y 383.391,Z 265.721,A -85,B 0,C 180,E1 17295.118,E2 17295.118} C_VEL
LIN {X 0,Y 380.512,Z 262.705,A -85,B 0,C 180,E1 17293.061,E2 17293.061} C_VEL
LIN {X 0,Y 379.113,Z 259.666,A -85,B 0,C 180,E1 17291.717,E2 17291.717} C_VEL
LIN {X 0,Y 375.9,Z 257.035,A -85,B 0,C 180,E1 17288.875,E2 17288.875} C_VEL
LIN {X 0,Y 374.343,Z 253.325,A -85,B 0,C 180,E1 17286.595,E2 17286.595} C_VEL
LIN {X 0,Y 370.867,Z 250.89,A -85,B 0,C 180,E1 17278.764,E2 17278.764} C_VEL
LIN {X 0,Y 371.49,Z 251.549,A -85,B 0,C 180,E1 17274.13,E2 17274.13} C_VEL
LIN {X 0,Y 374.488,Z 253.671,A -85,B 0,C 180,E1 17269.271,E2 17269.271} C_VEL
LIN {X 0,Y 376.122,Z 261.606,A -85,B 0,C 180,E1 17266.353,E2 17266.353} C_VEL
LIN {X 0,Y 378.615,Z 269.925,A -85,B 0,C 180,E1 17263.586,E2 17263.586} C_VEL
LIN {X 0,Y 385.424,Z 282.96,A -85,B 0,C 180,E1 17260.29,E2 17260.29} C_VEL
LIN {X 0,Y 393.512,Z 298.865,A -85,B 0,C 180,E1 17256.647,E2 17256.647} C_VEL
LIN {X 0,Y 402.331,Z 316.84,A -85,B 0,C 180,E1 17252.948,E2 17252.948} C_VEL
LIN {X 0,Y 410.157,Z 332.928,A -85,B 0,C 180,E1 17249.996,E2 17249.996} C_VEL
LIN {X 0,Y 428.238,Z 360.802,A -85,B 0,C 180,E1 17246.862,E2 17246.862} C_VEL
LIN {X 0,Y 436.471,Z 374.047,A -85,B 0,C 180,E1 17245.514,E2 17245.514} C_VEL
LIN {X 0,Y 417.243,Z 631.491,A -85,B 0,C 180,E1 17240.099,E2 17240.099} C_VEL
LIN {X 0,Y 412.894,Z 693.948,A -85,B 0,C 180,E1 17238.717,E2 17238.717} C_VEL
LIN {X 0,Y 410.167,Z 718.357,A -85,B 0,C 180,E1 17237.96,E2 17237.96} C_VEL
LIN {X 0,Y 406.626,Z 743.879,A -85,B 0,C 180,E1 17236.913,E2 17236.913} C_VEL
LIN {X 0,Y 402.884,Z 766.939,A -85,B 0,C 180,E1 17235.724,E2 17235.724} C_VEL
LIN {X 0,Y 398.654,Z 789.481,A -85,B 0,C 180,E1 17234.282,E2 17234.282} C_VEL
LIN {X 0,Y 393.831,Z 812.889,A -85,B 0,C 180,E1 17232.481,E2 17232.481} C_VEL
LIN {X 0,Y 389.308,Z 833.205,A -85,B 0,C 180,E1 17230.623,E2 17230.623} C_VEL
LIN {X 0,Y 384.718,Z 852.523,A -85,B 0,C 180,E1 17228.527,E2 17228.527} C_VEL
LIN {X 0,Y 380.138,Z 871.424,A -85,B 0,C 180,E1 17226.146,E2 17226.146} C_VEL
LIN {X 0,Y 375.883,Z 888.627,A -85,B 0,C 180,E1 17223.594,E2 17223.594} C_VEL
LIN {X 0,Y 371.678,Z 905.948,A -85,B 0,C 180,E1 17220.586,E2 17220.586} C_VEL
LIN {X 0,Y 368.526,Z 919.642,A -85,B 0,C 180,E1 17217.808,E2 17217.808} C_VEL
LIN {X 0,Y 365.762,Z 932.567,A -85,B 0,C 180,E1 17214.725,E2 17214.725} C_VEL
LIN {X 0,Y 363.603,Z 944.291,A -85,B 0,C 180,E1 17211.453,E2 17211.453} C_VEL
LIN {X 0,Y 362.169,Z 953.987,A -85,B 0,C 180,E1 17208.178,E2 17208.178} C_VEL
LIN {X 0,Y 361.326,Z 962.067,A -85,B 0,C 180,E1 17204.913,E2 17204.913} C_VEL
LIN {X 0,Y 360.957,Z 968.703,A -85,B 0,C 180,E1 17201.505,E2 17201.505} C_VEL
LIN {X 0,Y 360.949,Z 973.188,A -85,B 0,C 180,E1 17198.523,E2 17198.523} C_VEL
LIN {X 0,Y 361.102,Z 976.867,A -85,B 0,C 180,E1 17195.083,E2 17195.083} C_VEL
LIN {X 0,Y 361.251,Z 978.684,A -85,B 0,C 180,E1 17191.903,E2 17191.903} C_VEL
LIN {X 0,Y 361.231,Z 979.16,A -85,B 0,C 180,E1 17189.048,E2 17189.048} C_VEL
LIN {X 0,Y 361.074,Z 978.468,A -85,B 0,C 180,E1 17186.03,E2 17186.03} C_VEL
LIN {X 0,Y 360.804,Z 976.089,A -85,B 0,C 180,E1 17182.516,E2 17182.516} C_VEL
LIN {X 0,Y 360.711,Z 972.725,A -85,B 0,C 180,E1 17179.458,E2 17179.458} C_VEL
LIN {X 0,Y 360.927,Z 967.69,A -85,B 0,C 180,E1 17176.053,E2 17176.053} C_VEL
LIN {X 0,Y 361.857,Z 960.075,A -85,B 0,C 180,E1 17172.138,E2 17172.138} C_VEL
LIN {X 0,Y 363.44,Z 951.875,A -85,B 0,C 180,E1 17168.706,E2 17168.706} C_VEL
LIN {X 0,Y 366.317,Z 940.57,A -85,B 0,C 180,E1 17164.798,E2 17164.798} C_VEL
LIN {X 0,Y 370.299,Z 927.832,A -85,B 0,C 180,E1 17161.096,E2 17161.096} C_VEL
LIN {X 0,Y 375.296,Z 913.565,A -85,B 0,C 180,E1 17157.621,E2 17157.621} C_VEL
LIN {X 0,Y 381.882,Z 896.522,A -85,B 0,C 180,E1 17154.09,E2 17154.09} C_VEL
LIN {X 0,Y 389.169,Z 878.862,A -85,B 0,C 180,E1 17150.988,E2 17150.988} C_VEL
LIN {X 0,Y 397.276,Z 859.703,A -85,B 0,C 180,E1 17148.159,E2 17148.159} C_VEL
LIN {X 0,Y 406.471,Z 838.288,A -85,B 0,C 180,E1 17145.486,E2 17145.486} C_VEL
LIN {X 0,Y 416.369,Z 815.377,A -85,B 0,C 180,E1 17143.11,E2 17143.11} C_VEL
LIN {X 0,Y 425.924,Z 793.069,A -85,B 0,C 180,E1 17141.201,E2 17141.201} C_VEL
LIN {X 0,Y 435.049,Z 771.007,A -85,B 0,C 180,E1 17139.651,E2 17139.651} C_VEL
LIN {X 0,Y 443.884,Z 748.687,A -85,B 0,C 180,E1 17138.381,E2 17138.381} C_VEL
LIN {X 0,Y 448.557,Z 736.3,A -85,B 0,C 180,E1 17137.767,E2 17137.767} C_VEL
LIN {X 0,Y 438.455,Z 757.223,A -85,B 0,C 180,E1 17136.528,E2 17136.528} C_VEL
LIN {X 0,Y 428.026,Z 777.505,A -85,B 0,C 180,E1 17134.995,E2 17134.995} C_VEL
LIN {X 0,Y 417.47,Z 797.566,A -85,B 0,C 180,E1 17133.099,E2 17133.099} C_VEL
LIN {X 0,Y 407.438,Z 816.792,A -85,B 0,C 180,E1 17130.858,E2 17130.858} C_VEL
LIN {X 0,Y 398.353,Z 834.637,A -85,B 0,C 180,E1 17128.321,E2 17128.321} C_VEL
LIN {X 0,Y 390.604,Z 850.206,A -85,B 0,C 180,E1 17125.634,E2 17125.634} C_VEL
LIN {X 0,Y 384.339,Z 862.875,A -85,B 0,C 180,E1 17122.969,E2 17122.969} C_VEL
LIN {X 0,Y 379.023,Z 873.475,A -85,B 0,C 180,E1 17120.218,E2 17120.218} C_VEL
LIN {X 0,Y 374.57,Z 882.04,A -85,B 0,C 180,E1 17117.396,E2 17117.396} C_VEL
LIN {X 0,Y 370.918,Z 888.625,A -85,B 0,C 180,E1 17114.519,E2 17114.519} C_VEL
LIN {X 0,Y 368.15,Z 893.065,A -85,B 0,C 180,E1 17111.753,E2 17111.753} C_VEL
LIN {X 0,Y 366.013,Z 895.825,A -85,B 0,C 180,E1 17108.958,E2 17108.958} C_VEL
LIN {X 0,Y 364.426,Z 896.884,A -85,B 0,C 180,E1 17106.143,E2 17106.143} C_VEL
LIN {X 0,Y 363.265,Z 896.126,A -85,B 0,C 180,E1 17103.156,E2 17103.156} C_VEL
LIN {X 0,Y 362.594,Z 893.619,A -85,B 0,C 180,E1 17100.316,E2 17100.316} C_VEL
LIN {X 0,Y 362.254,Z 889.408,A -85,B 0,C 180,E1 17097.469,E2 17097.469} C_VEL
LIN {X 0,Y 362.232,Z 883.769,A -85,B 0,C 180,E1 17094.774,E2 17094.774} C_VEL
LIN {X 0,Y 362.532,Z 875.956,A -85,B 0,C 180,E1 17091.914,E2 17091.914} C_VEL
LIN {X 0,Y 363.206,Z 866.063,A -85,B 0,C 180,E1 17089.05,E2 17089.05} C_VEL
LIN {X 0,Y 364.27,Z 854.546,A -85,B 0,C 180,E1 17086.337,E2 17086.337} C_VEL
LIN {X 0,Y 365.672,Z 841.577,A -85,B 0,C 180,E1 17083.805,E2 17083.805} C_VEL
LIN {X 0,Y 367.459,Z 826.606,A -85,B 0,C 180,E1 17081.353,E2 17081.353} C_VEL
LIN {X 0,Y 369.541,Z 810.047,A -85,B 0,C 180,E1 17079.074,E2 17079.074} C_VEL
LIN {X 0,Y 371.846,Z 791.943,A -85,B 0,C 180,E1 17076.988,E2 17076.988} C_VEL
LIN {X 0,Y 374.252,Z 772.49,A -85,B 0,C 180,E1 17075.115,E2 17075.115} C_VEL
LIN {X 0,Y 376.791,Z 751.357,A -85,B 0,C 180,E1 17073.439,E2 17073.439} C_VEL
LIN {X 0,Y 379.246,Z 729.129,A -85,B 0,C 180,E1 17072.011,E2 17072.011} C_VEL
LIN {X 0,Y 381.469,Z 706.375,A -85,B 0,C 180,E1 17070.863,E2 17070.863} C_VEL
LIN {X 0,Y 383.428,Z 682.672,A -85,B 0,C 180,E1 17069.981,E2 17069.981} C_VEL
LIN {X 0,Y 395.248,Z 511.536,A -85,B 0,C 180,E1 17065.352,E2 17065.352} C_VEL
LIN {X 0,Y 391.838,Z 447.433,A -85,B 0,C 180,E1 17062.879,E2 17062.879} C_VEL
LIN {X 0,Y 393.218,Z 446.968,A -85,B 0,C 180,E1 17062.619,E2 17062.619} C_VEL
LIN {X 0,Y 395.398,Z 443.797,A -85,B 0,C 180,E1 17062.29,E2 17062.29} C_VEL
LIN {X 0,Y 398.815,Z 435.862,A -85,B 0,C 180,E1 17061.874,E2 17061.874} C_VEL
LIN {X 0,Y 400.426,Z 433.355,A -85,B 0,C 180,E1 17061.646,E2 17061.646} C_VEL
LIN {X 0,Y 404.177,Z 431.028,A -85,B 0,C 180,E1 17061.024,E2 17061.024} C_VEL
LIN {X 0,Y 408.609,Z 426.161,A -85,B 0,C 180,E1 17060.374,E2 17060.374} C_VEL
LIN {X 0,Y 409.577,Z 425.061,A -85,B 0,C 180,E1 17060.237,E2 17060.237} C_VEL
LIN {X 0,Y 414.152,Z 421.888,A -85,B 0,C 180,E1 17059.545,E2 17059.545} C_VEL
LIN {X 0,Y 418.92,Z 417.332,A -85,B 0,C 180,E1 17058.975,E2 17058.975} C_VEL
LIN {X 0,Y 423.934,Z 414.013,A -85,B 0,C 180,E1 17058.308,E2 17058.308} C_VEL
LIN {X 0,Y 428.557,Z 410.023,A -85,B 0,C 180,E1 17057.782,E2 17057.782} C_VEL
LIN {X 0,Y 431.714,Z 408.162,A -85,B 0,C 180,E1 17057.372,E2 17057.372} C_VEL
LIN {X 0,Y 430.489,Z 414.914,A -85,B 0,C 180,E1 17057.159,E2 17057.159} C_VEL
LIN {X 0,Y 425.936,Z 494.183,A -85,B 0,C 180,E1 17055.778,E2 17055.778} C_VEL
LIN {X 0,Y 421.205,Z 553.034,A -85,B 0,C 180,E1 17054.534,E2 17054.534} C_VEL
LIN {X 0,Y 415.261,Z 612.433,A -85,B 0,C 180,E1 17053.05,E2 17053.05} C_VEL
LIN {X 0,Y 410.707,Z 656.621,A -85,B 0,C 180,E1 17051.73,E2 17051.73} C_VEL
LIN {X 0,Y 408.041,Z 685.292,A -85,B 0,C 180,E1 17050.674,E2 17050.674} C_VEL
